# B&R Automation Studio project TD52 (part 56)

#### MsgEMCyclic.st - Cyclic code
```iecst
(*******************************************************************************
Msg_EM	 			 alarms generation MM_emission

This code is confidential and proprietary to the INNIO Company.
It may not be used in any form, or reproduced in any manner,
without written permission of the INNIO Company.
Copyright, INNIO Company, 2023

Customized modifications: -
------------------------

History:
-------
V0.01.0	02.11.2011	lettenb.	new
		27.05.2013	lettenb.	reset OUT_xx.txx2AB.bGnlTripx changed
V4.0.0  02-10-2013  Maxhera,    implementation of the module for modular software
V4.05.0	22.05.2017	Tinello		SCR added, 2276 deleted
		29.01.2018	Tinello		NOx warnings added
V4.05.1	19.02.2018	Tinello		9212 aktiviert, Verzögerung für MS-Sto von 60s auf 10s
V4.07.0	23.04.2019	Tinello		Neue Warnungen für NOx-Selbstdiagnose / Dosierung gestoppt / externe SCR Systeme / NOx lifetime reached
								Warning 2451, 2453 and 3456 can only be acknowledged if blocking of valve/pump is no longer present
								W3482, W3483 und A3380 deleted
V4.07.1	31.10.2019	Tinello		new parameter for lifetime monitoring / measurement signal error delay changed from 10s to 60s
V4.09.0	24.02.2020	Tinello		bugfix -> operating message was too short for HMI / SCR customer input always active
		01.07.2020	Tinello		bugfix -> Message only active if urea dosing controller is active
V4.11.0	11.04.2022	Tinello		CAT temp min monitoring added / W9252 delay from 0->5s
V4.13.0	21.11.2023	Tinello		New operating messages and warnings added
V4.14.0	18.06.2024	Soto	  	Low NOx sensor with CAN communication IF3 considered in W2609 (2023-183)

Instructions for use:
--------------------
1) declare alarm with function block "Alm"
	declare buffert alarm bit bMsg<message number>

2) use template to create a new alarm,
   substitue 0000 by alarm number and make settings:

	xMsg0000.Enable		:=	TRUE;		enable/disable alarm
	xMsg0000.Set		:=	FALSE;		alarm set condition
	xMsg0000.PT			:=	T#0s;		alarm delay time
	xMsg0000.Prio		:=	1;			alarm priority: 1-3 = trip, 4 = warning
	xMsg0000.RiskClass	:=	3;			risk class for remote alarm reset
	xMsg0000.Reset		:=	FALSE;		FALSE: for all standard alarms	prio 1,2,3 and warnings prio 4
										TRUE : for autoreset alarms

	bMsg0000			:=	xMsg0000.Q;	connect buffert alarm bit for VIS and control

3)  expand INIT

3)	include datapoint into OPC configuration for vis

Outstandings:
------------
(*******************************************************************************)
PROGRAM _CYCLIC

	(* reset general trip *)
	OUT_EM.tEM2AB.bGnlTrip1		:=	FALSE;
	OUT_EM.tEM2AB.bGnlTrip2		:=	FALSE;
	OUT_EM.tEM2AB.bGnlTrip3		:=	FALSE;
	OUT_EM.tEM2AB.bGnlWarning	:=	FALSE;
	OUT_EM.tEM2AB.bTriptype1	:=	FALSE;
	OUT_EM.tEM2AB.bTriptype2	:=	FALSE;
	OUT_EM.tEM2AB.bTriptype3	:=	FALSE;

	(* A2276 NOx deviation *) 					(* --> NOT USED *)
	xMsg2276.Enable	   	:= FALSE;
	xMsg2276.Set	   	:= FALSE;
	xMsg2276.PT		   	:= T#0s;
	xMsg2276.Prio 	   	:= 3;
	xMsg2276.RiskClass 	:= 4;
	xMsg2276.Reset		:= FALSE;
	xMsg2276();
	MM2VIS.bMsg2276   	:= xMsg2276.Q;

	(* W2446 SCR BUS communication interrupted *)
	xMsg2446.Enable		:= TRUE;
	xMsg2446.Set		:= bAMM_2446;
	xMsg2446.PT			:= T#10s;
	xMsg2446.Prio		:= 4;
	xMsg2446.RiskClass	:= 4;
	xMsg2446.Reset		:= FALSE;
	xMsg2446();
	MM2VIS.bMsg2446		:= xMsg2446.Q;

	(* W2447 SCR Measuring signal failure urea pressure before dosing *)
	xMsg2447.Enable		:= TRUE;
	xMsg2447.Set		:= bAMM_2447;
	xMsg2447.PT			:= T#10s;
	xMsg2447.Prio		:= 4;
	xMsg2447.RiskClass	:= 4;
	xMsg2447.Reset		:= FALSE;
	xMsg2447();
	MM2VIS.bMsg2447		:= xMsg2447.Q;

	(* W2448 SCR Urea pressure before dosing minimum *)
	xMsg2448.Enable		:= TRUE;
	xMsg2448.Set		:= bAMM_2448;
	xMsg2448.PT			:= T#60s;
	xMsg2448.Prio		:= 4;
	xMsg2448.RiskClass	:= 4;
	xMsg2448.Reset		:= FALSE;
	xMsg2448();
	MM2VIS.bMsg2448		:= xMsg2448.Q;

	(* W2449 SCR Urea pressure before dosing maximum *)
	xMsg2449.Enable		:= TRUE;
	xMsg2449.Set		:= bAMM_2449;
	xMsg2449.PT			:= T#60s;
	xMsg2449.Prio		:= 4;
	xMsg2449.RiskClass	:= 4;
	xMsg2449.Reset		:= FALSE;
	xMsg2449();
	MM2VIS.bMsg2449		:= xMsg2449.Q;

	(* W2450 SCR Leakage in urea dosing cabinet *)
	xMsg2450.Enable		:= Para.bSCR_Active OR Para.bSCR_Cust_Active;
	xMsg2450.Set		:= NOT IN_EM.tLev_SCR_UreaDosingCabinet_Hi.Di;
	xMsg2450.PT			:= T#30s;
	xMsg2450.Prio		:= 4;
	xMsg2450.RiskClass	:= 4;
	xMsg2450.Reset		:= FALSE;
	xMsg2450();
	MM2VIS.bMsg2450		:= xMsg2450.Q;

	(* W2451 SCR Urea dosing valve - error *)
	xMsg2451.Enable		:= TRUE;
	xMsg2451.Set		:= bAMM_2451 OR (MM2VIS.bMsg2451 AND (VIS2MM.bSCR_UreaDosingUnit_Blocked OR
															  VIS2MM.bSCR_UreaDosingUnit2_Blocked  ));
	xMsg2451.PT			:= T#1s;
	xMsg2451.Prio		:= 4;
	xMsg2451.RiskClass	:= 4;
	xMsg2451.Reset		:= FALSE;
	xMsg2451();
	MM2VIS.bMsg2451		:= xMsg2451.Q;

	(* W2452 SCR Measuring signal failure urea flow rate after dosing *)
	xMsg2452.Enable		:= TRUE;
	xMsg2452.Set		:= bAMM_2452;
	xMsg2452.PT			:= T#10s;
	xMsg2452.Prio		:= 4;
	xMsg2452.RiskClass	:= 4;
	xMsg2452.Reset		:= FALSE;
	xMsg2452();
	MM2VIS.bMsg2452		:= xMsg2452.Q;

	(* W2453 SCR Urea flow rate - valve characteristic deviating maximum *)
	xMsg2453.Enable		:= TRUE;
	xMsg2453.Set		:= bAMM_2453 OR (MM2VIS.bMsg2453 AND (VIS2MM.bSCR_UreaDosingUnit_Blocked OR
															  VIS2MM.bSCR_UreaDosingUnit2_Blocked  ));
	xMsg2453.PT			:= T#1s;
	xMsg2453.Prio		:= 4;
	xMsg2453.RiskClass	:= 4;
	xMsg2453.Reset		:= FALSE;
	xMsg2453();
	MM2VIS.bMsg2453		:= xMsg2453.Q;

	(* W2454 SCR Compressed air supply pressure urea injection maximum *)
	xMsg2454.Enable		:= TRUE;
	xMsg2454.Set		:= bAMM_2454;
	xMsg2454.PT			:= T#60s;
	xMsg2454.Prio		:= 4;
	xMsg2454.RiskClass	:= 4;
	xMsg2454.Reset		:= FALSE;
	xMsg2454();
	MM2VIS.bMsg2454		:= xMsg2454.Q;

	(* W2455 SCR Deviation to continous emission monitoring system maximum *)
	xMsg2455.Enable		:= TRUE;
	xMsg2455.Set		:= (EDGEPOS(bAMM_2455_CO) OR EDGEPOS(bAMM_2455_NOx) OR EDGEPOS(bAMM_2455_NOxS)) AND xTON_bRel_SCR_UDC_5m.Q;
	xMsg2455.PT			:= T#0s;
	xMsg2455.Prio		:= 4;
	xMsg2455.RiskClass	:= 4;
	xMsg2455.Reset		:= FALSE;
	xMsg2455();
	MM2VIS.bMsg2455		:= xMsg2455.Q;

	(* W2456 SCR Emission measurement line 1 - O2 maximum *)
	xMsg2456.Enable		:= TRUE;
	xMsg2456.Set		:= bAMM_2456;
	xMsg2456.PT			:= T#60s;
	xMsg2456.Prio		:= 4;
	xMsg2456.RiskClass	:= 4;
	xMsg2456.Reset		:= FALSE;
	xMsg2456();
	MM2VIS.bMsg2456		:= xMsg2456.Q;

	(* W2457 SCR Measuring signal failure emission measurement line 1 - O2 sensor *)
	xMsg2457.Enable		:= TRUE;
	xMsg2457.Set		:= bAMM_2457;
	xMsg2457.PT			:= T#10s;
	xMsg2457.Prio		:= 4;
	xMsg2457.RiskClass	:= 4;
	xMsg2457.Reset		:= FALSE;
	xMsg2457();
	MM2VIS.bMsg2457		:= xMsg2457.Q;

	(* W2458 SCR Measuring signal failure emission measurement line 2 - NO2 sensor *)
	xMsg2458.Enable		:= TRUE;
	xMsg2458.Set		:= bAMM_2458;
	xMsg2458.PT			:= T#10s;
	xMsg2458.Prio		:= 4;
	xMsg2458.RiskClass	:= 4;
	xMsg2458.Reset		:= FALSE;
	xMsg2458();
	MM2VIS.bMsg2458		:= xMsg2458.Q;

	(* W2464 SCR Urea dosing unit (external) - error *)
	xMsg2464.Enable		:= TRUE;
	xMsg2464.Set		:= bAMM_2464;
	xMsg2464.PT			:= T#5s;
	xMsg2464.Prio		:= 4;
	xMsg2464.RiskClass	:= 4;
	xMsg2464.Reset		:= FALSE;
	xMsg2464();
	MM2VIS.bMsg2464		:= xMsg2464.Q;

	(* W2607 CAN failure - NOx sensor CAN interface 1 *)
	xMsg2607.Enable	   	:= TRUE;
	xMsg2607.Set	   	:= bAMM_NOxS_CAN_IF1;
	xMsg2607.PT		   	:= T#10s;
	xMsg2607.Prio 	   	:= 4;
	xMsg2607.RiskClass 	:= 4;
	xMsg2607();
	MM2VIS.bMsg2607    	:= xMsg2607.Q;

	(* W2609 CAN failure - NOx sensor CAN interface 2 or 3 *)
	xMsg2609.Enable	   	:= TRUE;
	xMsg2609.Set	   	:= bAMM_NOxS_CAN_IF2 OR bAMM_NOxS_CAN_IF3;
	xMsg2609.PT		   	:= T#10s;
	xMsg2609.Prio 	   	:= 4;
	xMsg2609.RiskClass 	:= 4;
	xMsg2609();
	MM2VIS.bMsg2609    	:= xMsg2609.Q;

	(* W2610 No connection to the sensor - NOx sensor engine out *)
	xMsg2610.Enable	   	:= TRUE;
	xMsg2610.Set	   	:= bAMM_NOxS_CAN_EngOut;
	xMsg2610.PT		   	:= T#1s;
	xMsg2610.Prio 	   	:= 4;
	xMsg2610.RiskClass 	:= 4;
	xMsg2610();
	MM2VIS.bMsg2610   	:= xMsg2610.Q;

	(* W2697 SCR Urea dosing unit - maintenance needed *)
	xMsg2697.Enable		:= TRUE;
	xMsg2697.Set		:= bAMM_2697;
	xMsg2697.PT			:= T#0s;
	xMsg2697.Prio		:= 4;
	xMsg2697.RiskClass	:= 4;
	xMsg2697.Reset		:= FALSE;
	xMsg2697();
	MM2VIS.bMsg2697		:= xMsg2697.Q;

	(* W2766 Catalyst temperature minimum *)
	xMsg2766.Enable		:= TRUE;
	xMsg2766.Set		:= bAMM_2766;
	xMsg2766.PT			:= T#10s;
	xMsg2766.Prio		:= 4;
	xMsg2766.RiskClass	:= 4;
	xMsg2766.Reset		:= FALSE;
	xMsg2766();
	MM2VIS.bMsg2766		:= xMsg2766.Q;

	(* W2769 SCR Emission measurement air line - moisture maximum *)
	xMsg2769.Enable		:= TRUE;
	xMsg2769.Set		:= bAMM_2769;
	xMsg2769.PT			:= T#0s;
	xMsg2769.Prio		:= 4;
	xMsg2769.RiskClass	:= 4;
	xMsg2769.Reset		:= FALSE;
	xMsg2769();
	MM2VIS.bMsg2769		:= xMsg2769.Q;

	(* A3379 SCR Exhaust temperatures CAT maximum *)
		xTON_T_SCR_Cat3(IN:= NOT IN_EM.tT_SCR_Cat_HiHi.Di, PT:= T#1s);

	xMsg3379.Enable		:= TRUE;
	xMsg3379.Set		:= bAMM_3379 OR xTON_T_SCR_Cat3.Q;
	xMsg3379.PT			:= T#0s;
	xMsg3379.Prio		:= 3;
	xMsg3379.RiskClass	:= 4;
	xMsg3379.Reset		:= FALSE;
	xMsg3379();
	MM2VIS.bMsg3379		:= xMsg3379.Q;

	(* A3380 SCR CO emission average maximum *)			(* --> NOT USED *)
	xMsg3380.Enable		:= FALSE;
	xMsg3380.Set		:= FALSE;
	xMsg3380.PT			:= T#0s;
	xMsg3380.Prio		:= 3;
	xMsg3380.RiskClass	:= 4;
	xMsg3380.Reset		:= FALSE;
	xMsg3380();
	MM2VIS.bMsg3380		:= xMsg3380.Q;

	(* A3381 NOx emissions - short-term average high *)
	xMsg3381.Enable		:= TRUE;
	xMsg3381.Set		:= bAMM_3381;
	xMsg3381.PT			:= T#0s;
	xMsg3381.Prio		:= 3;
	xMsg3381.RiskClass	:= 4;
	xMsg3381.Reset		:= FALSE;
	xMsg3381();
	MM2VIS.bMsg3381		:= xMsg3381.Q;

	(* A3383 SCR Measuring signal failure exhaust temperatures CAT *)
	xMsg3383.Enable		:= TRUE;
	xMsg3383.Set		:= bAMM_3383;
	xMsg3383.PT			:= T#300s;
	xMsg3383.Prio		:= 3;
	xMsg3383.RiskClass	:= 4;
	xMsg3383.Reset		:= FALSE;
	xMsg3383();
	MM2VIS.bMsg3383		:= xMsg3383.Q;

	(*	W3450 SCR Group alarm - exhaust after treatment system *)	(* --> NOT USED *)
	xMsg3450.Enable 	:= FALSE;
	xMsg3450.Set 		:= FALSE;
	xMsg3450.PT			:= T#0s;
	xMsg3450.Prio		:= 4;
	xMsg3450.RiskClass	:= 4;
	xMsg3450();
	MM2VIS.bMsg3450		:= xMsg3450.Q;

	(* W3451 SCR Power supply to the valves interrupted *)
	xMsg3451.Enable		:= TRUE;
	xMsg3451.Set		:= bAMM_3451;
	xMsg3451.PT			:= T#10s;
	xMsg3451.Prio		:= 4;
	xMsg3451.RiskClass	:= 4;
	xMsg3451.Reset		:= FALSE;
	xMsg3451();
	MM2VIS.bMsg3451		:= xMsg3451.Q;

	(* W3452 SCR Measuring signal failure urea pressure after dosing *)
	xMsg3452.Enable		:= TRUE;
	xMsg3452.Set		:= bAMM_3452;
	xMsg3452.PT			:= T#10s;
	xMsg3452.Prio		:= 4;
	xMsg3452.RiskClass	:= 4;
	xMsg3452.Reset		:= FALSE;
	xMsg3452();
	MM2VIS.bMsg3452		:= xMsg3452.Q;

	(* W3453 SCR Urea pressure after dosing maximum *)
	xMsg3453.Enable		:= TRUE;
	xMsg3453.Set		:= bAMM_3453;
	xMsg3453.PT			:= T#0s;
	xMsg3453.Prio		:= 4;
	xMsg3453.RiskClass	:= 4;
	xMsg3453.Reset		:= FALSE;
	xMsg3453();
	MM2VIS.bMsg3453		:= xMsg3453.Q;

	(* W3454 SCR Urea pressure after dosing minimum *)
	xMsg3454.Enable		:= TRUE;
	xMsg3454.Set		:= bAMM_3454;
	xMsg3454.PT			:= T#60s;
	xMsg3454.Prio		:= 4;
	xMsg3454.RiskClass	:= 4;
	xMsg3454.Reset		:= FALSE;
	xMsg3454();
	MM2VIS.bMsg3454		:= xMsg3454.Q;

	(* W3455 SCR Urea flow rate after dosing maximum *)
	xMsg3455.Enable		:= TRUE;
	xMsg3455.Set		:= bAMM_3455;
	xMsg3455.PT			:= T#600s;
	xMsg3455.Prio		:= 4;
	xMsg3455.RiskClass	:= 4;
	xMsg3455.Reset		:= FALSE;
	xMsg3455();
	MM2VIS.bMsg3455		:= xMsg3455.Q;

	(* W3456 SCR Urea dosing pump - error *)
	xMsg3456.Enable		:= TRUE;
	xMsg3456.Set		:= bAMM_3456 OR (MM2VIS.bMsg3456 AND (VIS2MM.bSCR_UreaDosingUnit_Blocked OR
															  VIS2MM.bSCR_UreaDosingUnit2_Blocked  ));
	xMsg3456.PT			:= T#1s;
	xMsg3456.Prio		:= 4;
	xMsg3456.RiskClass	:= 4;
	xMsg3456.Reset		:= FALSE;
	xMsg3456();
	MM2VIS.bMsg3456		:= xMsg3456.Q;

	(* W3457 SCR Urea-air valve blocked *)
	xMsg3457.Enable		:= TRUE;
	xMsg3457.Set		:= bAMM_3457;
	xMsg3457.PT			:= T#45s;
	xMsg3457.Prio		:= 4;
	xMsg3457.RiskClass	:= 4;
	xMsg3457.Reset		:= FALSE;
	xMsg3457();
	MM2VIS.bMsg3457		:= xMsg3457.Q;

	(* W3458 SCR Urea tank level minimum *)
	xMsg3458.Enable		:= Para.bSCR_Active OR Para.bSCR_Cust_Active;
	xMsg3458.Set		:= NOT IN_EM.tLev_SCR_UreaTank_Lo.Di OR (Para.bLev_SCR_UreaTank_Exist AND NOT bAMM_9379 AND IN_EM.tLev_SCR_UreaTank.Ai < Para.rLev_SCR_UreaTank_Lo);
	xMsg3458.PT			:= T#300s;
	xMsg3458.Prio		:= 4;
	xMsg3458.RiskClass	:= 4;
	xMsg3458.Reset		:= FALSE;
	xMsg3458();
	MM2VIS.bMsg3458		:= xMsg3458.Q;

	(* W3459 SCR Urea tank level minimum - dosing deactivated *)
	xMsg3459.Enable		:= TRUE;
	xMsg3459.Set		:= bAMM_3459;
	xMsg3459.PT			:= T#0s;
	xMsg3459.Prio		:= 4;
	xMsg3459.RiskClass	:= 4;
	xMsg3459.Reset		:= FALSE;
	xMsg3459();
	MM2VIS.bMsg3459		:= xMsg3459.Q;

	(* W3460 SCR Urea supply pump not operating *)
	xMsg3460.Enable		:= TRUE;
	xMsg3460.Set		:= bAMM_3460;
	xMsg3460.PT			:= T#30s;
	xMsg3460.Prio		:= 4;
	xMsg3460.RiskClass	:= 4;
	xMsg3460.Reset		:= FALSE;
	xMsg3460();
	MM2VIS.bMsg3460		:= xMsg3460.Q;

	(* W3461 SCR Measuring signal failure compressed air supply pressure urea injection *)
	xMsg3461.Enable		:= TRUE;
	xMsg3461.Set		:= bAMM_3461;
	xMsg3461.PT			:= T#10s;
	xMsg3461.Prio		:= 4;
	xMsg3461.RiskClass	:= 4;
	xMsg3461.Reset		:= FALSE;
	xMsg3461();
	MM2VIS.bMsg3461		:= xMsg3461.Q;

	(* W3462 SCR Compressed air supply pressure urea injection minimum *)
	xMsg3462.Enable		:= TRUE;
	xMsg3462.Set		:= bAMM_3462;
	xMsg3462.PT			:= T#60s;
	xMsg3462.Prio		:= 4;
	xMsg3462.RiskClass	:= 4;
	xMsg3462.Reset		:= FALSE;
	xMsg3462();
	MM2VIS.bMsg3462		:= xMsg3462.Q;

	(* W3463 SCR Compressed air urea injection power supply interrupted *)
	xMsg3463.Enable		:= TRUE;
	xMsg3463.Set		:= bAMM_3463;
	xMsg3463.PT			:= T#10s;
	xMsg3463.Prio		:= 4;
	xMsg3463.RiskClass	:= 4;
	xMsg3463.Reset		:= FALSE;
	xMsg3463();
	MM2VIS.bMsg3463		:= xMsg3463.Q;

	(* W3464 SCR Measuring signal failure exhaust pressure CAT inlet *)
	xMsg3464.Enable		:= TRUE;
	xMsg3464.Set		:= bAMM_3464;
	xMsg3464.PT			:= T#10s;
	xMsg3464.Prio		:= 4;
	xMsg3464.RiskClass	:= 4;
	xMsg3464.Reset		:= FALSE;
	xMsg3464();
	MM2VIS.bMsg3464		:= xMsg3464.Q;

	(* W3465 SCR Measuring signal failure exhaust pressure CAT outlet *)
	xMsg3465.Enable		:= TRUE;
	xMsg3465.Set		:= bAMM_3465;
	xMsg3465.PT			:= T#10s;
	xMsg3465.Prio		:= 4;
	xMsg3465.RiskClass	:= 4;
	xMsg3465.Reset		:= FALSE;
	xMsg3465();
	MM2VIS.bMsg3465		:= xMsg3465.Q;

	(* W3466 SCR Measuring signal failure exhaust temperature CAT inlet *)
	xMsg3466.Enable		:= TRUE;
	xMsg3466.Set		:= bAMM_3466;
	xMsg3466.PT			:= T#10s;
	xMsg3466.Prio		:= 4;
	xMsg3466.RiskClass	:= 4;
	xMsg3466.Reset		:= FALSE;
	xMsg3466();
	MM2VIS.bMsg3466		:= xMsg3466.Q;

	(* W3467 SCR Measuring signal failure exhaust temperature CAT outlet *)
	xMsg3467.Enable		:= TRUE;
	xMsg3467.Set		:= bAMM_3467;
	xMsg3467.PT			:= T#10s;
	xMsg3467.Prio		:= 4;
	xMsg3467.RiskClass	:= 4;
	xMsg3467.Reset		:= FALSE;
	xMsg3467();
	MM2VIS.bMsg3467		:= xMsg3467.Q;

	(* W3469 SCR Exhaust differential pressure CAT maximum *)
	xMsg3469.Enable		:= TRUE;
	xMsg3469.Set		:= bAMM_3469;
	xMsg3469.PT			:= T#300s;
	xMsg3469.Prio		:= 4;
	xMsg3469.RiskClass	:= 4;
	xMsg3469.Reset		:= FALSE;
	xMsg3469();
	MM2VIS.bMsg3469		:= xMsg3469.Q;

	(* W3470 SCR Emission measurement sample gas cooler - error *)
	xMsg3470.Enable		:= TRUE;
	xMsg3470.Set		:= bAMM_3470;
	xMsg3470.PT			:= T#60s;
	xMsg3470.Prio		:= 4;
	xMsg3470.RiskClass	:= 4;
	xMsg3470.Reset		:= FALSE;
	xMsg3470();
	MM2VIS.bMsg3470		:= xMsg3470.Q;

	(* W3471 SCR Emission measurement line 1 - sample gas pump not ready *)
	xMsg3471.Enable		:= TRUE;
	xMsg3471.Set		:= bAMM_3471;
	xMsg3471.PT			:= T#10s;
	xMsg3471.Prio		:= 4;
	xMsg3471.RiskClass	:= 4;
	xMsg3471.Reset		:= FALSE;
	xMsg3471();
	MM2VIS.bMsg3471		:= xMsg3471.Q;

	(* W3472 SCR Emission measurement line 2 - sample gas pump not operating *)
	xMsg3472.Enable		:= TRUE;
	xMsg3472.Set		:= bAMM_3472;
	xMsg3472.PT			:= T#10s;
	xMsg3472.Prio		:= 4;
	xMsg3472.RiskClass	:= 4;
	xMsg3472.Reset		:= FALSE;
	xMsg3472();
	MM2VIS.bMsg3472		:= xMsg3472.Q;

	(* W3473 SCR Emission measurement line 1 - moisture maximum *)
	xMsg3473.Enable		:= TRUE;
	xMsg3473.Set		:= bAMM_3473;
	xMsg3473.PT			:= T#10s;
	xMsg3473.Prio		:= 4;
	xMsg3473.RiskClass	:= 4;
	xMsg3473.Reset		:= FALSE;
	xMsg3473();
	MM2VIS.bMsg3473		:= xMsg3473.Q;

	(* W3474 SCR Emission measurement line 2 - moisture maximum *)
	xMsg3474.Enable		:= TRUE;
	xMsg3474.Set		:= bAMM_3474;
	xMsg3474.PT			:= T#10s;
	xMsg3474.Prio		:= 4;
	xMsg3474.RiskClass	:= 4;
	xMsg3474.Reset		:= FALSE;
	xMsg3474();
	MM2VIS.bMsg3474		:= xMsg3474.Q;

	(* W3475 SCR Emission measurement line 1 - flow rate minimum *)
	xMsg3475.Enable		:= TRUE;
	xMsg3475.Set		:= bAMM_3475;
	xMsg3475.PT			:= T#10s;
	xMsg3475.Prio		:= 4;
	xMsg3475.RiskClass	:= 4;
	xMsg3475.Reset		:= FALSE;
	xMsg3475();
	MM2VIS.bMsg3475		:= xMsg3475.Q;

	(* W3476 SCR Emission measurement line 2 - flow rate minimum *)
	xMsg3476.Enable		:= TRUE;
	xMsg3476.Set		:= bAMM_3476;
	xMsg3476.PT			:= T#10s;
	xMsg3476.Prio		:= 4;
	xMsg3476.RiskClass	:= 4;
	xMsg3476.Reset		:= FALSE;
	xMsg3476();
	MM2VIS.bMsg3476		:= xMsg3476.Q;

	(* W3477 SCR Measuring signal failure emission measurement line 2 - NO sensor *)
	xMsg3477.Enable		:= TRUE;
	xMsg3477.Set		:= bAMM_3477;
	xMsg3477.PT			:= T#10s;
	xMsg3477.Prio		:= 4;
	xMsg3477.RiskClass	:= 4;
	xMsg3477.Reset		:= FALSE;
	xMsg3477();
	MM2VIS.bMsg3477		:= xMsg3477.Q;

	(* W3478 SCR Measuring signal failure emission measurement line 1 - NO sensor *)
	xMsg3478.Enable		:= TRUE;
	xMsg3478.Set		:= bAMM_3478;
	xMsg3478.PT			:= T#10s;
	xMsg3478.Prio		:= 4;
	xMsg3478.RiskClass	:= 4;
	xMsg3478.Reset		:= FALSE;
	xMsg3478();
	MM2VIS.bMsg3478		:= xMsg3478.Q;

	(* W3479 SCR Measuring signal failure emission measurement line 1 - NO2 sensor *)
	xMsg3479.Enable		:= TRUE;
	xMsg3479.Set		:= bAMM_3479;
	xMsg3479.PT			:= T#10s;
	xMsg3479.Prio		:= 4;
	xMsg3479.RiskClass	:= 4;
	xMsg3479.Reset		:= FALSE;
	xMsg3479();
	MM2VIS.bMsg3479		:= xMsg3479.Q;

	(* W3480 SCR NH3 slip detection deactivated *)
	xMsg3480.Enable		:= TRUE;
	xMsg3480.Set		:= bAMM_3480;
	xMsg3480.PT			:= T#0s;
	xMsg3480.Prio		:= 4;
	xMsg3480.RiskClass	:= 4;
	xMsg3480.Reset		:= FALSE;
	xMsg3480();
	MM2VIS.bMsg3480		:= xMsg3480.Q;

	(* W3481 SCR Measuring signal failure emission measurement line 1 - CO sensor *)
	xMsg3481.Enable		:= TRUE;
	xMsg3481.Set		:= bAMM_3481;
	xMsg3481.PT			:= T#10s;
	xMsg3481.Prio		:= 4;
	xMsg3481.RiskClass	:= 4;
	xMsg3481.Reset		:= FALSE;
	xMsg3481();
	MM2VIS.bMsg3481		:= xMsg3481.Q;

	(* W3482 SCR NOx emission to check *)				(* --> NOT USED *)
	xMsg3482.Enable		:= FALSE;
	xMsg3482.Set		:= FALSE;
	xMsg3482.PT			:= T#0s;
	xMsg3482.Prio		:= 4;
	xMsg3482.RiskClass	:= 4;
	xMsg3482.Reset		:= FALSE;
	xMsg3482();
	MM2VIS.bMsg3482		:= xMsg3482.Q;

	(* W3483 SCR CO emission to check *)				(* --> NOT USED *)
	xMsg3483.Enable		:= FALSE;
	xMsg3483.Set		:= FALSE;
	xMsg3483.PT			:= T#0s;
	xMsg3483.Prio		:= 4;
	xMsg3483.RiskClass	:= 4;
	xMsg3483.Reset		:= FALSE;
	xMsg3483();
	MM2VIS.bMsg3483		:= xMsg3483.Q;

	(* W3484 CO emissions - short-term average high *)
	xMsg3484.Enable		:= TRUE;
	xMsg3484.Set		:= bAMM_3484;
	xMsg3484.PT			:= T#0s;
	xMsg3484.Prio		:= 4;
	xMsg3484.RiskClass	:= 4;
	xMsg3484.Reset		:= FALSE;
	xMsg3484();
	MM2VIS.bMsg3484		:= xMsg3484.Q;

	(* W3485 NOx emissions - short-term average high *)
	xMsg3485.Enable		:= TRUE;
	xMsg3485.Set		:= bAMM_3485;
	xMsg3485.PT			:= T#0s;
	xMsg3485.Prio		:= 4;
	xMsg3485.RiskClass	:= 4;
	xMsg3485.Reset		:= FALSE;
	xMsg3485();
	MM2VIS.bMsg3485		:= xMsg3485.Q;

	(* W3486 SCR Urea flow rate after dosing minimum *)
	xMsg3486.Enable		:= TRUE;
	xMsg3486.Set		:= bAMM_3486;
	xMsg3486.PT			:= T#600s;
	xMsg3486.Prio		:= 4;
	xMsg3486.RiskClass	:= 4;
	xMsg3486.Reset		:= FALSE;
	xMsg3486();
	MM2VIS.bMsg3486		:= xMsg3486.Q;

	(* W3487 SCR Exhaust temperature CAT inlet maximum *)
	xMsg3487.Enable		:= TRUE;
	xMsg3487.Set		:= bAMM_3487;
	xMsg3487.PT			:= T#10s;
	xMsg3487.Prio		:= 4;
	xMsg3487.RiskClass	:= 4;
	xMsg3487.Reset		:= FALSE;
	xMsg3487();
	MM2VIS.bMsg3487		:= xMsg3487.Q;

	(* W3488 SCR Exhaust temperature CAT outlet maximum *)
	xMsg3488.Enable		:= TRUE;
	xMsg3488.Set		:= bAMM_3488;
	xMsg3488.PT			:= T#10s;
	xMsg3488.Prio		:= 4;
	xMsg3488.RiskClass	:= 4;
	xMsg3488.Reset		:= FALSE;
	xMsg3488();
	MM2VIS.bMsg3488		:= xMsg3488.Q;

	(* W3489 SCR Emergency Stop SCR control cabinet *)		(* --> NOT USED	*)
	xMsg3489.Enable 	:= FALSE;
	xMsg3489.Set 		:= FALSE;
	xMsg3489.PT			:= T#0s;
	xMsg3489.Prio		:= 4;
	xMsg3489.RiskClass	:= 4;
	xMsg3489.Reset		:= FALSE;
	xMsg3489();
	MM2VIS.bMsg3489		:= xMsg3489.Q;

	(* W9201 Measuring signal failure O2, NOx sensor engine out *)
	xMsg9201.Enable 	:= TRUE;
	xMsg9201.Set 		:= bAMM_O2_NOxS_EngOut_Ms;
	xMsg9201.PT			:= T#60s;
	xMsg9201.Prio		:= 4;
	xMsg9201.RiskClass	:= 4;
	xMsg9201.Reset		:= FALSE;
	xMsg9201();
	MM2VIS.bMsg9201		:= xMsg9201.Q;

	(* W9202 Measuring signal failure NOx, NOx sensor engine out *)
	xMsg9202.Enable 	:= TRUE;
	xMsg9202.Set 		:= bAMM_NOx_NOxS_EngOut_Ms;
	xMsg9202.PT			:= T#60s;
	xMsg9202.Prio		:= 4;
	xMsg9202.RiskClass	:= 4;
	xMsg9202.Reset		:= FALSE;
	xMsg9202();
	MM2VIS.bMsg9202		:= xMsg9202.Q;

	(* W9203 No connection to the sensor - NOx sensor engine out A *)
	xMsg9203.Enable 	:= TRUE;
	xMsg9203.Set 		:= bAMM_NOxS_CAN_EngOut_A;
	xMsg9203.PT			:= T#1s;
	xMsg9203.Prio		:= 4;
	xMsg9203.RiskClass	:= 4;
	xMsg9203.Reset		:= FALSE;
	xMsg9203();
	MM2VIS.bMsg9203		:= xMsg9203.Q;

	(* W9204 Measuring signal failure O2, NOx sensor engine out – bank A *)
	xMsg9204.Enable 	:= TRUE;
	xMsg9204.Set 		:= bAMM_O2_NOxS_EngOut_A_Ms;
	xMsg9204.PT			:= T#60s;
	xMsg9204.Prio		:= 4;
	xMsg9204.RiskClass	:= 4;
	xMsg9204.Reset		:= FALSE;
	xMsg9204();
	MM2VIS.bMsg9204		:= xMsg9204.Q;

	(* W9205 Measuring signal failure NOx, NOx sensor engine out – bank A *)
	xMsg9205.Enable 	:= TRUE;
	xMsg9205.Set 		:= bAMM_NOx_NOxS_EngOut_A_Ms;
	xMsg9205.PT			:= T#60s;
	xMsg9205.Prio		:= 4;
	xMsg9205.RiskClass	:= 4;
	xMsg9205.Reset		:= FALSE;
	xMsg9205();
	MM2VIS.bMsg9205		:= xMsg9205.Q;

	(* W9206 No connection to the sensor - NOx sensor engine out B *)
	xMsg9206.Enable 	:= TRUE;
	xMsg9206.Set 		:= bAMM_NOxS_CAN_EngOut_B;
	xMsg9206.PT			:= T#1s;
	xMsg9206.Prio		:= 4;
	xMsg9206.RiskClass	:= 4;
	xMsg9206.Reset		:= FALSE;
	xMsg9206();
	MM2VIS.bMsg9206		:= xMsg9206.Q;

	(* W9207 Measuring signal failure O2, NOx sensor engine out – bank B *)
	xMsg9207.Enable 	:= TRUE;
	xMsg9207.Set 		:= bAMM_O2_NOxS_EngOut_B_Ms;
	xMsg9207.PT			:= T#60s;
	xMsg9207.Prio		:= 4;
	xMsg9207.RiskClass	:= 4;
	xMsg9207.Reset		:= FALSE;
	xMsg9207();
	MM2VIS.bMsg9207		:= xMsg9207.Q;

	(* W9208 Measuring signal failure NOx, NOx sensor engine out – bank B *)
	xMsg9208.Enable 	:= TRUE;
	xMsg9208.Set 		:= bAMM_NOx_NOxS_EngOut_B_Ms;
	xMsg9208.PT			:= T#60s;
	xMsg9208.Prio		:= 4;
	xMsg9208.RiskClass	:= 4;
	xMsg9208.Reset		:= FALSE;
	xMsg9208();
	MM2VIS.bMsg9208		:= xMsg9208.Q;

	(* W9209 No connection to the sensor - NOx sensor CAT out *)
	xMsg9209.Enable 	:= TRUE;
	xMsg9209.Set 		:= bAMM_NOxS_CAN_CatOut;
	xMsg9209.PT			:= T#1s;
	xMsg9209.Prio		:= 4;
	xMsg9209.RiskClass	:= 4;
	xMsg9209.Reset		:= FALSE;
	xMsg9209();
	MM2VIS.bMsg9209		:= xMsg9209.Q;

	(* W9210 Measuring signal failure O2, NOx sensor CAT out *)
	xMsg9210.Enable 	:= TRUE;
	xMsg9210.Set 		:= bAMM_O2_NOxS_CatOut_Ms;
	xMsg9210.PT			:= T#60s;
	xMsg9210.Prio		:= 4;
	xMsg9210.RiskClass	:= 4;
	xMsg9210.Reset		:= FALSE;
	xMsg9210();
	MM2VIS.bMsg9210		:= xMsg9210.Q;

	(* W9211 Measuring signal failure NOx, NOx sensor CAT out *)
	xMsg9211.Enable 	:= TRUE;
	xMsg9211.Set 		:= bAMM_NOx_NOxS_CatOut_Ms;
	xMsg9211.PT			:= T#60s;
	xMsg9211.Prio		:= 4;
	xMsg9211.RiskClass	:= 4;
	xMsg9211.Reset		:= FALSE;
	xMsg9211();
	MM2VIS.bMsg9211		:= xMsg9211.Q;

	(* W9212 SCR Air compressor - maintenance needed  *)
	xMsg9212.Enable 	:= TRUE;
	xMsg9212.Set 		:= bAMM_9212;
	xMsg9212.PT			:= T#0s;
	xMsg9212.Prio		:= 4;
	xMsg9212.RiskClass	:= 4;
	xMsg9212.Reset		:= FALSE;
	xMsg9212();
	MM2VIS.bMsg9212		:= xMsg9212.Q;

	(* W9233 Lifetime reached - NOx sensor engine out *)
	xMsg9233.Enable 	:= TRUE;
	xMsg9233.Set 		:= bNOxS_EngOut_Exist 	AND MM2VIS.iNOxS_EngOut_OpHours   >= Para.iNOxS_Lifetime;
	xMsg9233.PT			:= T#0s;
	xMsg9233.Prio		:= 4;
	xMsg9233.RiskClass	:= 4;
	xMsg9233.Reset		:= FALSE;
	xMsg9233();
	MM2VIS.bMsg9233		:= xMsg9233.Q;

	(* W9234 Lifetime reached - NOx sensor engine out A *)
	xMsg9234.Enable 	:= TRUE;
	xMsg9234.Set 		:= bNOxS_EngOut_A_Exist AND MM2VIS.iNOxS_EngOut_A_OpHours >= Para.iNOxS_Lifetime;
	xMsg9234.PT			:= T#0s;
	xMsg9234.Prio		:= 4;
	xMsg9234.RiskClass	:= 4;
	xMsg9234.Reset		:= FALSE;
	xMsg9234();
	MM2VIS.bMsg9234		:= xMsg9234.Q;

	(* W9235 Lifetime reached - NOx sensor engine out B *)
	xMsg9235.Enable 	:= TRUE;
	xMsg9235.Set 		:= bNOxS_EngOut_B_Exist	AND MM2VIS.iNOxS_EngOut_B_OpHours >= Para.iNOxS_Lifetime;
	xMsg9235.PT			:= T#0s;
	xMsg9235.Prio		:= 4;
	xMsg9235.RiskClass	:= 4;
	xMsg9235.Reset		:= FALSE;
	xMsg9235();
	MM2VIS.bMsg9235		:= xMsg9235.Q;

	(* W9236 Lifetime reached - NOx sensor CAT out *)
	xMsg9236.Enable 	:= TRUE;
	xMsg9236.Set 		:= bNOxS_CatOut_Exist 	AND MM2VIS.iNOxS_CatOut_OpHours   >= Para.iNOxS_Lifetime;
	xMsg9236.PT			:= T#0s;
	xMsg9236.Prio		:= 4;
	xMsg9236.RiskClass	:= 4;
	xMsg9236.Reset		:= FALSE;
	xMsg9236();
	MM2VIS.bMsg9236		:= xMsg9236.Q;

	(* W9250 O2 deviation bank A/B maximum - NOx sensor engine out *)
	xMsg9250.Enable 	:= TRUE;
	xMsg9250.Set 		:= bAMM_O2_NOxS_EngOut_Dev_Hi;
	xMsg9250.PT			:= T#0s;
	xMsg9250.Prio		:= 4;
	xMsg9250.RiskClass	:= 4;
	xMsg9250.Reset		:= FALSE;
	xMsg9250();
	MM2VIS.bMsg9250		:= xMsg9250.Q;

	(* W9251 NOx deviation bank A/B maximum - NOx sensor engine out *)
	xMsg9251.Enable 	:= TRUE;
	xMsg9251.Set 		:= bAMM_NOx_NOxS_EngOut_Dev_Hi;
	xMsg9251.PT			:= T#0s;
	xMsg9251.Prio		:= 4;
	xMsg9251.RiskClass	:= 4;
	xMsg9251.Reset		:= FALSE;
	xMsg9251();
	MM2VIS.bMsg9251		:= xMsg9251.Q;

	(* W9252 NOx emissions - daily average high *)
	xMsg9252.Enable 	:= TRUE;
	xMsg9252.Set 		:= bAMM_NOx_Em_AvgDaily_Hi;
	xMsg9252.PT			:= T#5s;
	xMsg9252.Prio		:= 4;
	xMsg9252.RiskClass	:= 4;
	xMsg9252.Reset		:= FALSE;
	xMsg9252();
	MM2VIS.bMsg9252		:= xMsg9252.Q;

	(* W9277 SCR Urea dosing stopped - error *)
	xMsg9277.Enable 	:= TRUE;
	xMsg9277.Set 		:= bAMM_9277;
	xMsg9277.PT			:= T#0s;
	xMsg9277.Prio		:= 4;
	xMsg9277.RiskClass	:= 4;
	xMsg9277.Reset		:= FALSE;
	xMsg9277();
	MM2VIS.bMsg9277		:= xMsg9277.Q;

	(* W9278 SCR Catalyst - failure (DI from customer) *)
	xMsg9278.Enable 	:= TRUE;
	xMsg9278.Set 		:= NOT IN_EM.tSCR_Catalyst_Rdy.Di;
	xMsg9278.PT			:= T#1s;
	xMsg9278.Prio		:= 4;
	xMsg9278.RiskClass	:= 4;
	xMsg9278.Reset		:= FALSE;
	xMsg9278();
	MM2VIS.bMsg9278		:= xMsg9278.Q;

	(* W9379 SCR Measuring signal failure urea tank level *)
	xMsg9379.Enable 	:= TRUE;
	xMsg9379.Set 		:= bAMM_9379;
	xMsg9379.PT			:= T#10s;
	xMsg9379.Prio		:= 4;
	xMsg9379.RiskClass	:= 4;
	xMsg9379.Reset		:= FALSE;
	xMsg9379();
	MM2VIS.bMsg9379		:= xMsg9379.Q;

	(* W9380 SCR Urea flow dosing error *)
	xMsg9380.Enable 	:= TRUE;
	xMsg9380.Set 		:= bAMM_9380;
	xMsg9380.PT			:= T#0s;
	xMsg9380.Prio		:= 4;
	xMsg9380.RiskClass	:= 4;
	xMsg9380.Reset		:= FALSE;
	xMsg9380();
	MM2VIS.bMsg9380		:= xMsg9380.Q;

	(*---------------------------------------------------------------------------*)
	(* operating messages > AMM *)

	(* B2877 SCR Exhaust after treatment deactivated *)	(* --> NOT USED *)
	xMsg2877.Enable 	:= FALSE;
	xMsg2877.Set 		:= FALSE;
	xMsg2877.Reset     	:= TRUE;
	xMsg2877();
	MM2VIS.bMsg2877		:= xMsg2877.Q;

	(* B2878 SCR Urea dosing activated *)
	xMsg2878.Enable		:= TRUE;
	xMsg2878.Set		:= bOpM_2878;
	xMsg2878.Reset		:= TRUE;
	xMsg2878();
	MM2VIS.bMsg2878		:= xMsg2878.Q;

	(* B2879 SCR Urea dosing deactivated *)
	xMsg2879.Enable		:= TRUE;
	xMsg2879.Set		:= bOpM_2879;
	xMsg2879.Reset		:= TRUE;
	xMsg2879();
	MM2VIS.bMsg2879		:= xMsg2879.Q;

	(* B2884 SCR Manual mode on *)
	xMsg2884.Enable		:= TRUE;
	xMsg2884.Set		:= bOpM_2884;
	xMsg2884.Reset		:= TRUE;
	xMsg2884();
	MM2VIS.bMsg2884		:= xMsg2884.Q;

	(* B2885 SCR Manual mode off *)
	xMsg2885.Enable		:= TRUE;
	xMsg2885.Set		:= bOpM_2885;
	xMsg2885.Reset		:= TRUE;
	xMsg2885();
	MM2VIS.bMsg2885		:= xMsg2885.Q;

	(* B2923 SCR NH3 slip detection started *)
	xMsg2923.Enable		:= TRUE;
	xMsg2923.Set		:= bOpM_2923;
	xMsg2923.Reset		:= TRUE;
	xMsg2923();
	MM2VIS.bMsg2923		:= xMsg2923.Q;

	(* B2924 SCR NH3 slip detection completed *)
	xMsg2924.Enable		:= TRUE;
	xMsg2924.Set		:= bOpM_2924;
	xMsg2924.Reset		:= TRUE;
	xMsg2924();
	MM2VIS.bMsg2924		:= xMsg2924.Q;

	(* B2971 Error during self-diagnosis - NOx sensor engine out *)
	xTOF_EngOut_DiagErr(IN 	:= bOpM_NOxS_EngOut_DiagErr, 	PT := T#1s);		(* increase message time from 100ms to 1s for HMI *)

	xMsg2971.Enable			:= TRUE;
	xMsg2971.Set			:= xTOF_EngOut_DiagErr.Q;
	xMsg2971.Reset			:= TRUE;
	xMsg2971();
	MM2VIS.bMsg2971			:= xMsg2971.Q;

	(* B2974 Error during self-diagnosis - NOx sensor engine out A *)
	xTOF_EngOut_A_DiagErr(IN:= bOpM_NOxS_EngOut_A_DiagErr, 	PT := T#1s);		(* increase message time from 100ms to 1s for HMI *)

	xMsg2974.Enable			:= TRUE;
	xMsg2974.Set			:= xTOF_EngOut_A_DiagErr.Q;
	xMsg2974.Reset			:= TRUE;
	xMsg2974();
	MM2VIS.bMsg2974			:= xMsg2974.Q;

	(* B2977 Error during self-diagnosis - NOx sensor engine out B *)
	xTOF_EngOut_B_DiagErr(IN:= bOpM_NOxS_EngOut_B_DiagErr, 	PT := T#1s);		(* increase message time from 100ms to 1s for HMI *)

	xMsg2977.Enable			:= TRUE;
	xMsg2977.Set			:= xTOF_EngOut_B_DiagErr.Q;
	xMsg2977.Reset			:= TRUE;
	xMsg2977();
	MM2VIS.bMsg2977			:= xMsg2977.Q;

	(* B2980 Error during self-diagnosis - NOx sensor CAT out *)
	xTOF_CatOut_DiagErr(IN 	:= bOpM_NOxS_CatOut_DiagErr, 	PT := T#1s);		(* increase message time from 100ms to 1s for HMI *)

	xMsg2980.Enable			:= TRUE;
	xMsg2980.Set			:= xTOF_CatOut_DiagErr.Q;
	xMsg2980.Reset			:= TRUE;
	xMsg2980();
	MM2VIS.bMsg2980			:= xMsg2980.Q;

	(* B9077 SCR NH3 slip detection interrupted *)
	xMsg9077.Enable			:= TRUE;
	xMsg9077.Set			:= bOpM_9077;
	xMsg9077.Reset			:= TRUE;
	xMsg9077();
	MM2VIS.bMsg9077			:= xMsg9077.Q;

	(* B9079 SCR Urea dosing - dosing conditions reached *)
	xMsg9079.Enable			:= TRUE;
	xMsg9079.Set			:= bOpM_9079;
	xMsg9079.Reset			:= TRUE;
	xMsg9079();
	MM2VIS.bMsg9079			:= xMsg9079.Q;

	(* B9080 SCR Urea dosing - dosing conditions ended *)
	xMsg9080.Enable			:= TRUE;
	xMsg9080.Set			:= bOpM_9080;
	xMsg9080.Reset			:= TRUE;
	xMsg9080();
	MM2VIS.bMsg9080			:= xMsg9080.Q;

	(* B9081 SCR Urea dosing - requested *)
	xMsg9081.Enable			:= TRUE;
	xMsg9081.Set			:= bOpM_9081;
	xMsg9081.Reset			:= TRUE;
	xMsg9081();
	MM2VIS.bMsg9081			:= xMsg9081.Q;

	(* B9082 SCR Urea dosing - unrequested *)
	xMsg9082.Enable			:= TRUE;
	xMsg9082.Set			:= bOpM_9082;
	xMsg9082.Reset			:= TRUE;
	xMsg9082();
	MM2VIS.bMsg9082			:= xMsg9082.Q;

	(*--------------------------------------------------------------------------*)
	(* general alarms for further module operations *)
	bGnlTrip1	:= OUT_EM.tEM2AB.bGnlTrip1   OR IN_EM.tAB2EM.bGnlTrip1;
	bGnlTrip2	:= OUT_EM.tEM2AB.bGnlTrip2   OR IN_EM.tAB2EM.bGnlTrip2;
	bGnlTrip3	:= OUT_EM.tEM2AB.bGnlTrip3   OR IN_EM.tAB2EM.bGnlTrip3;
	bGnlWarning	:= OUT_EM.tEM2AB.bGnlWarning OR IN_EM.tAB2EM.bGnlWarning;

	bGnlTrip	:=	bGnlTrip1 OR bGnlTrip2 OR bGnlTrip3;

	(*******************************************************************************)
END_PROGRAM
```

#### MsgEMInit.st - Initial code
```iecst
(*******************************************************************************
Msg_EM	 			 alarms generation MM_emission

This code is confidential and proprietary to the INNIO Company.
It may not be used in any form, or reproduced in any manner,
without written permission of the INNIO Company.
Copyright, INNIO Company, 2019

Customized modifications: -
------------------------

History:
-------
V0.00.0	29.07.2011	lettenb.	new
V4.00.0 22-08-2013  Maxhera,    implementation of the module for modular software
V4.05.0	22.05.2017	Tinello		SCR added
		29.01.2018	Tinello		NOx warnings added

Instructions for use:
--------------------
1) declare alarm with function block "Msg"

2) use template to create a new alarm, substitue 0000 by message number:

	xMsg0000.Num		:=	0000;					alarm number
	xMsg0000.AmmSysAdr	:=  iAdrAmmBase2MM;			do not change
	xMsg0000.AmmOutAdr	:=  iAdrMM2AmmBase;			do not change

3) 	set alarm number

Outstandings:
------------
(*******************************************************************************)
PROGRAM _INIT

	iAdrAmmBase2MM		:=  ADR(IN_EM.tAB2EM);
	iAdrMM2AmmBase		:=  ADR(OUT_EM.tEM2AB);

	xMsg2276.Num		:= 2276;
	xMsg2276.AmmInAdr	:=  iAdrAmmBase2MM;
	xMsg2276.AmmOutAdr	:=  iAdrMM2AmmBase;

	xMsg2446.Num		:= 2446;
	xMsg2446.AmmInAdr	:= iAdrAmmBase2MM;
	xMsg2446.AmmOutAdr	:= iAdrMM2AmmBase;

	xMsg2447.Num		:= 2447;
	xMsg2447.AmmInAdr	:= iAdrAmmBase2MM;
	xMsg2447.AmmOutAdr	:= iAdrMM2AmmBase;

	xMsg2448.Num		:= 2448;
	xMsg2448.AmmInAdr	:= iAdrAmmBase2MM;
	xMsg2448.AmmOutAdr	:= iAdrMM2AmmBase;

	xMsg2449.Num		:= 2449;
	xMsg2449.AmmInAdr	:= iAdrAmmBase2MM;
	xMsg2449.AmmOutAdr	:= iAdrMM2AmmBase;

	xMsg2450.Num		:= 2450;
	xMsg2450.AmmInAdr	:= iAdrAmmBase2MM;
	xMsg2450.AmmOutAdr	:= iAdrMM2AmmBase;

	xMsg2451.Num		:= 2451;
	xMsg2451.AmmInAdr	:= iAdrAmmBase2MM;
	xMsg2451.AmmOutAdr	:= iAdrMM2AmmBase;

	xMsg2452.Num		:= 2452;
	xMsg2452.AmmInAdr	:= iAdrAmmBase2MM;
	xMsg2452.AmmOutAdr	:= iAdrMM2AmmBase;

	xMsg2453.Num		:= 2453;
	xMsg2453.AmmInAdr	:= iAdrAmmBase2MM;
	xMsg2453.AmmOutAdr	:= iAdrMM2AmmBase;

	xMsg2454.Num		:= 2454;
	xMsg2454.AmmInAdr	:= iAdrAmmBase2MM;
	xMsg2454.AmmOutAdr	:= iAdrMM2AmmBase;

	xMsg2455.Num		:= 2455;
	xMsg2455.AmmInAdr	:= iAdrAmmBase2MM;
	xMsg2455.AmmOutAdr	:= iAdrMM2AmmBase;

	xMsg2456.Num		:= 2456;
	xMsg2456.AmmInAdr	:= iAdrAmmBase2MM;
	xMsg2456.AmmOutAdr	:= iAdrMM2AmmBase;

	xMsg2457.Num		:= 2457;
	xMsg2457.AmmInAdr	:= iAdrAmmBase2MM;
	xMsg2457.AmmOutAdr	:= iAdrMM2AmmBase;

	xMsg2458.Num		:= 2458;
	xMsg2458.AmmInAdr	:= iAdrAmmBase2MM;
	xMsg2458.AmmOutAdr	:= iAdrMM2AmmBase;

	xMsg2464.Num		:= 2464;
	xMsg2464.AmmInAdr	:= iAdrAmmBase2MM;
	xMsg2464.AmmOutAdr	:= iAdrMM2AmmBase;

	xMsg2607.Num		:= 2607;
	xMsg2607.AmmInAdr	:= iAdrAmmBase2MM;
	xMsg2607.AmmOutAdr	:= iAdrMM2AmmBase;

	xMsg2609.Num		:= 2609;
	xMsg2609.AmmInAdr	:= iAdrAmmBase2MM;
	xMsg2609.AmmOutAdr	:=  iAdrMM2AmmBase;

	xMsg2610.Num		:= 2610;
	xMsg2610.AmmInAdr	:=  iAdrAmmBase2MM;
	xMsg2610.AmmOutAdr	:=  iAdrMM2AmmBase;

	xMsg2697.Num		:=	2697;
	xMsg2697.AmmInAdr	:=  iAdrAmmBase2MM;
	xMsg2697.AmmOutAdr	:=  iAdrMM2AmmBase;

	xMsg2766.Num		:=	2766;
	xMsg2766.AmmInAdr	:=  iAdrAmmBase2MM;
	xMsg2766.AmmOutAdr	:=  iAdrMM2AmmBase;

	xMsg2769.Num		:=	2769;
	xMsg2769.AmmInAdr	:=  iAdrAmmBase2MM;
	xMsg2769.AmmOutAdr	:=  iAdrMM2AmmBase;

	xMsg2877.Num 		:= 2877;
	xMsg2877.AmmInAdr	:= iAdrAmmBase2MM;
	xMsg2877.AmmOutAdr	:= iAdrMM2AmmBase;

	xMsg2878.Num 		:= 2878;
	xMsg2878.AmmInAdr	:= iAdrAmmBase2MM;
	xMsg2878.AmmOutAdr	:= iAdrMM2AmmBase;

	xMsg2879.Num 		:= 2879;
	xMsg2879.AmmInAdr	:= iAdrAmmBase2MM;
	xMsg2879.AmmOutAdr	:= iAdrMM2AmmBase;

	xMsg2884.Num 		:= 2884;
	xMsg2884.AmmInAdr	:= iAdrAmmBase2MM;
	xMsg2884.AmmOutAdr	:= iAdrMM2AmmBase;

	xMsg2885.Num 		:= 2885;
	xMsg2885.AmmInAdr	:= iAdrAmmBase2MM;
	xMsg2885.AmmOutAdr	:= iAdrMM2AmmBase;

	xMsg2923.Num 		:= 2923;
	xMsg2923.AmmInAdr	:= iAdrAmmBase2MM;
	xMsg2923.AmmOutAdr	:= iAdrMM2AmmBase;

	xMsg2924.Num 		:= 2924;
	xMsg2924.AmmInAdr	:= iAdrAmmBase2MM;
	xMsg2924.AmmOutAdr	:= iAdrMM2AmmBase;

	xMsg2971.Num 		:= 2971;
	xMsg2971.AmmInAdr	:= iAdrAmmBase2MM;
	xMsg2971.AmmOutAdr	:= iAdrMM2AmmBase;

	xMsg2974.Num 		:= 2974;
	xMsg2974.AmmInAdr	:= iAdrAmmBase2MM;
	xMsg2974.AmmOutAdr	:= iAdrMM2AmmBase;

	xMsg2977.Num 		:= 2977;
	xMsg2977.AmmInAdr	:= iAdrAmmBase2MM;
	xMsg2977.AmmOutAdr	:= iAdrMM2AmmBase;

	xMsg2980.Num 		:= 2980;
	xMsg2980.AmmInAdr	:= iAdrAmmBase2MM;
	xMsg2980.AmmOutAdr	:= iAdrMM2AmmBase;

	xMsg3379.Num 		:= 3379;
	xMsg3379.AmmInAdr	:= iAdrAmmBase2MM;
	xMsg3379.AmmOutAdr	:= iAdrMM2AmmBase;

	xMsg3380.Num 		:= 3380;
	xMsg3380.AmmInAdr	:= iAdrAmmBase2MM;
	xMsg3380.AmmOutAdr	:= iAdrMM2AmmBase;

	xMsg3381.Num 		:= 3381;
	xMsg3381.AmmInAdr	:= iAdrAmmBase2MM;
	xMsg3381.AmmOutAdr	:= iAdrMM2AmmBase;

	xMsg3383.Num 		:= 3383;
	xMsg3383.AmmInAdr	:= iAdrAmmBase2MM;
	xMsg3383.AmmOutAdr	:= iAdrMM2AmmBase;

	xMsg3450.Num 		:= 3450;
	xMsg3450.AmmInAdr	:= iAdrAmmBase2MM;
	xMsg3450.AmmOutAdr	:= iAdrMM2AmmBase;

	xMsg3451.Num 		:= 3451;
	xMsg3451.AmmInAdr	:= iAdrAmmBase2MM;
	xMsg3451.AmmOutAdr	:= iAdrMM2AmmBase;

	xMsg3452.Num 		:= 3452;
	xMsg3452.AmmInAdr	:= iAdrAmmBase2MM;
	xMsg3452.AmmOutAdr	:= iAdrMM2AmmBase;

	xMsg3453.Num 		:= 3453;
	xMsg3453.AmmInAdr	:= iAdrAmmBase2MM;
	xMsg3453.AmmOutAdr	:= iAdrMM2AmmBase;

	xMsg3454.Num 		:= 3454;
	xMsg3454.AmmInAdr	:= iAdrAmmBase2MM;
	xMsg3454.AmmOutAdr	:= iAdrMM2AmmBase;

	xMsg3455.Num 		:= 3455;
	xMsg3455.AmmInAdr	:= iAdrAmmBase2MM;
	xMsg3455.AmmOutAdr	:= iAdrMM2AmmBase;

	xMsg3456.Num 		:= 3456;
	xMsg3456.AmmInAdr	:= iAdrAmmBase2MM;
	xMsg3456.AmmOutAdr	:= iAdrMM2AmmBase;

	xMsg3457.Num 		:= 3457;
	xMsg3457.AmmInAdr	:= iAdrAmmBase2MM;
	xMsg3457.AmmOutAdr	:= iAdrMM2AmmBase;

	xMsg3458.Num 		:= 3458;
	xMsg3458.AmmInAdr	:= iAdrAmmBase2MM;
	xMsg3458.AmmOutAdr	:= iAdrMM2AmmBase;

	xMsg3459.Num 		:= 3459;
	xMsg3459.AmmInAdr	:= iAdrAmmBase2MM;
	xMsg3459.AmmOutAdr	:= iAdrMM2AmmBase;

	xMsg3460.Num 		:= 3460;
	xMsg3460.AmmInAdr	:= iAdrAmmBase2MM;
	xMsg3460.AmmOutAdr	:= iAdrMM2AmmBase;

	xMsg3461.Num 		:= 3461;
	xMsg3461.AmmInAdr	:= iAdrAmmBase2MM;
	xMsg3461.AmmOutAdr	:= iAdrMM2AmmBase;

	xMsg3462.Num 		:= 3462;
	xMsg3462.AmmInAdr	:= iAdrAmmBase2MM;
	xMsg3462.AmmOutAdr	:= iAdrMM2AmmBase;

	xMsg3463.Num 		:= 3463;
	xMsg3463.AmmInAdr	:= iAdrAmmBase2MM;
	xMsg3463.AmmOutAdr	:= iAdrMM2AmmBase;

	xMsg3464.Num 		:= 3464;
	xMsg3464.AmmInAdr	:= iAdrAmmBase2MM;
	xMsg3464.AmmOutAdr	:= iAdrMM2AmmBase;

	xMsg3465.Num 		:= 3465;
	xMsg3465.AmmInAdr	:= iAdrAmmBase2MM;
	xMsg3465.AmmOutAdr	:= iAdrMM2AmmBase;

	xMsg3466.Num 		:= 3466;
	xMsg3466.AmmInAdr	:= iAdrAmmBase2MM;
	xMsg3466.AmmOutAdr	:= iAdrMM2AmmBase;

	xMsg3467.Num 		:= 3467;
	xMsg3467.AmmInAdr	:= iAdrAmmBase2MM;
	xMsg3467.AmmOutAdr	:= iAdrMM2AmmBase;

	xMsg3469.Num 		:= 3469;
	xMsg3469.AmmInAdr	:= iAdrAmmBase2MM;
	xMsg3469.AmmOutAdr	:= iAdrMM2AmmBase;

	xMsg3470.Num 		:= 3470;
	xMsg3470.AmmInAdr	:= iAdrAmmBase2MM;
	xMsg3470.AmmOutAdr	:= iAdrMM2AmmBase;

	xMsg3471.Num 		:= 3471;
	xMsg3471.AmmInAdr	:= iAdrAmmBase2MM;
	xMsg3471.AmmOutAdr	:= iAdrMM2AmmBase;

	xMsg3472.Num 		:= 3472;
	xMsg3472.AmmInAdr	:= iAdrAmmBase2MM;
	xMsg3472.AmmOutAdr	:= iAdrMM2AmmBase;

	xMsg3473.Num 		:= 3473;
	xMsg3473.AmmInAdr	:= iAdrAmmBase2MM;
	xMsg3473.AmmOutAdr	:= iAdrMM2AmmBase;

	xMsg3474.Num 		:= 3474;
	xMsg3474.AmmInAdr	:= iAdrAmmBase2MM;
	xMsg3474.AmmOutAdr	:= iAdrMM2AmmBase;

	xMsg3475.Num 		:= 3475;
	xMsg3475.AmmInAdr	:= iAdrAmmBase2MM;
	xMsg3475.AmmOutAdr	:= iAdrMM2AmmBase;

	xMsg3476.Num 		:= 3476;
	xMsg3476.AmmInAdr	:= iAdrAmmBase2MM;
	xMsg3476.AmmOutAdr	:= iAdrMM2AmmBase;

	xMsg3477.Num 		:= 3477;
	xMsg3477.AmmInAdr	:= iAdrAmmBase2MM;
	xMsg3477.AmmOutAdr	:= iAdrMM2AmmBase;

	xMsg3478.Num 		:= 3478;
	xMsg3478.AmmInAdr	:= iAdrAmmBase2MM;
	xMsg3478.AmmOutAdr	:= iAdrMM2AmmBase;

	xMsg3479.Num 		:= 3479;
	xMsg3479.AmmInAdr	:= iAdrAmmBase2MM;
	xMsg3479.AmmOutAdr	:= iAdrMM2AmmBase;

	xMsg3480.Num 		:= 3480;
	xMsg3480.AmmInAdr	:= iAdrAmmBase2MM;
	xMsg3480.AmmOutAdr	:= iAdrMM2AmmBase;

	xMsg3481.Num 		:= 3481;
	xMsg3481.AmmInAdr	:= iAdrAmmBase2MM;
	xMsg3481.AmmOutAdr	:= iAdrMM2AmmBase;

	xMsg3482.Num 		:= 3482;
	xMsg3482.AmmInAdr	:= iAdrAmmBase2MM;
	xMsg3482.AmmOutAdr	:= iAdrMM2AmmBase;

	xMsg3483.Num 		:= 3483;
	xMsg3483.AmmInAdr	:= iAdrAmmBase2MM;
	xMsg3483.AmmOutAdr	:= iAdrMM2AmmBase;

	xMsg3484.Num 		:= 3484;
	xMsg3484.AmmInAdr	:= iAdrAmmBase2MM;
	xMsg3484.AmmOutAdr	:= iAdrMM2AmmBase;

	xMsg3485.Num 		:= 3485;
	xMsg3485.AmmInAdr	:= iAdrAmmBase2MM;
	xMsg3485.AmmOutAdr	:= iAdrMM2AmmBase;

	xMsg3486.Num 		:= 3486;
	xMsg3486.AmmInAdr	:= iAdrAmmBase2MM;
	xMsg3486.AmmOutAdr	:= iAdrMM2AmmBase;

	xMsg3487.Num 		:= 3487;
	xMsg3487.AmmInAdr	:= iAdrAmmBase2MM;
	xMsg3487.AmmOutAdr	:= iAdrMM2AmmBase;

	xMsg3488.Num 		:= 3488;
	xMsg3488.AmmInAdr	:= iAdrAmmBase2MM;
	xMsg3488.AmmOutAdr	:= iAdrMM2AmmBase;

	xMsg3489.Num 		:= 3489;
	xMsg3489.AmmInAdr	:= iAdrAmmBase2MM;
	xMsg3489.AmmOutAdr	:= iAdrMM2AmmBase;

	xMsg9077.Num 		:= 9077;
	xMsg9077.AmmInAdr	:= iAdrAmmBase2MM;
	xMsg9077.AmmOutAdr	:= iAdrMM2AmmBase;

	xMsg9079.Num 		:= 9079;
	xMsg9079.AmmInAdr	:= iAdrAmmBase2MM;
	xMsg9079.AmmOutAdr	:= iAdrMM2AmmBase;

	xMsg9080.Num 		:= 9080;
	xMsg9080.AmmInAdr	:= iAdrAmmBase2MM;
	xMsg9080.AmmOutAdr	:= iAdrMM2AmmBase;

	xMsg9081.Num 		:= 9081;
	xMsg9081.AmmInAdr	:= iAdrAmmBase2MM;
	xMsg9081.AmmOutAdr	:= iAdrMM2AmmBase;

	xMsg9082.Num 		:= 9082;
	xMsg9082.AmmInAdr	:= iAdrAmmBase2MM;
	xMsg9082.AmmOutAdr	:= iAdrMM2AmmBase;

	xMsg9201.Num 		:= 9201;
	xMsg9201.AmmInAdr	:= iAdrAmmBase2MM;
	xMsg9201.AmmOutAdr	:= iAdrMM2AmmBase;

	xMsg9202.Num 		:= 9202;
	xMsg9202.AmmInAdr	:= iAdrAmmBase2MM;
	xMsg9202.AmmOutAdr	:= iAdrMM2AmmBase;

	xMsg9203.Num 		:= 9203;
	xMsg9203.AmmInAdr	:= iAdrAmmBase2MM;
	xMsg9203.AmmOutAdr	:= iAdrMM2AmmBase;

	xMsg9204.Num 		:= 9204;
	xMsg9204.AmmInAdr	:= iAdrAmmBase2MM;
	xMsg9204.AmmOutAdr	:= iAdrMM2AmmBase;

	xMsg9205.Num 		:= 9205;
	xMsg9205.AmmInAdr	:= iAdrAmmBase2MM;
	xMsg9205.AmmOutAdr	:= iAdrMM2AmmBase;

	xMsg9206.Num 		:= 9206;
	xMsg9206.AmmInAdr	:= iAdrAmmBase2MM;
	xMsg9206.AmmOutAdr	:= iAdrMM2AmmBase;

	xMsg9207.Num 		:= 9207;
	xMsg9207.AmmInAdr	:= iAdrAmmBase2MM;
	xMsg9207.AmmOutAdr	:= iAdrMM2AmmBase;

	xMsg9208.Num 		:= 9208;
	xMsg9208.AmmInAdr	:= iAdrAmmBase2MM;
	xMsg9208.AmmOutAdr	:= iAdrMM2AmmBase;

	xMsg9209.Num 		:= 9209;
	xMsg9209.AmmInAdr	:= iAdrAmmBase2MM;
	xMsg9209.AmmOutAdr	:= iAdrMM2AmmBase;

	xMsg9210.Num 		:= 9210;
	xMsg9210.AmmInAdr	:= iAdrAmmBase2MM;
	xMsg9210.AmmOutAdr	:= iAdrMM2AmmBase;

	xMsg9211.Num 		:= 9211;
	xMsg9211.AmmInAdr	:= iAdrAmmBase2MM;
	xMsg9211.AmmOutAdr	:= iAdrMM2AmmBase;

	xMsg9212.Num 		:= 9212;
	xMsg9212.AmmInAdr	:= iAdrAmmBase2MM;
	xMsg9212.AmmOutAdr	:= iAdrMM2AmmBase;

	xMsg9233.Num 		:= 9233;
	xMsg9233.AmmInAdr	:= iAdrAmmBase2MM;
	xMsg9233.AmmOutAdr	:= iAdrMM2AmmBase;

	xMsg9234.Num 		:= 9234;
	xMsg9234.AmmInAdr	:= iAdrAmmBase2MM;
	xMsg9234.AmmOutAdr	:= iAdrMM2AmmBase;

	xMsg9235.Num 		:= 9235;
	xMsg9235.AmmInAdr	:= iAdrAmmBase2MM;
	xMsg9235.AmmOutAdr	:= iAdrMM2AmmBase;

	xMsg9236.Num 		:= 9236;
	xMsg9236.AmmInAdr	:= iAdrAmmBase2MM;
	xMsg9236.AmmOutAdr	:= iAdrMM2AmmBase;

	xMsg9250.Num 		:= 9250;
	xMsg9250.AmmInAdr	:= iAdrAmmBase2MM;
	xMsg9250.AmmOutAdr	:= iAdrMM2AmmBase;

	xMsg9251.Num 		:= 9251;
	xMsg9251.AmmInAdr	:= iAdrAmmBase2MM;
	xMsg9251.AmmOutAdr	:= iAdrMM2AmmBase;

	xMsg9252.Num 		:= 9252;
	xMsg9252.AmmInAdr	:= iAdrAmmBase2MM;
	xMsg9252.AmmOutAdr	:= iAdrMM2AmmBase;

	xMsg9277.Num 		:= 9277;
	xMsg9277.AmmInAdr	:= iAdrAmmBase2MM;
	xMsg9277.AmmOutAdr	:= iAdrMM2AmmBase;

	xMsg9278.Num 		:= 9278;
	xMsg9278.AmmInAdr	:= iAdrAmmBase2MM;
	xMsg9278.AmmOutAdr	:= iAdrMM2AmmBase;

	xMsg9379.Num 		:= 9379;
	xMsg9379.AmmInAdr	:= iAdrAmmBase2MM;
	xMsg9379.AmmOutAdr	:= iAdrMM2AmmBase;

	xMsg9380.Num 		:= 9380;
	xMsg9380.AmmInAdr	:= iAdrAmmBase2MM;
	xMsg9380.AmmOutAdr	:= iAdrMM2AmmBase;
END_PROGRAM
```

#### MsgEM.var - Local variables
```iecst
VAR
	iAdrAmmBase2MM : UDINT;
	iAdrMM2AmmBase : UDINT;
	xMsg2276 : Msg; (*NOx deviation --> canceled*)
	xMsg2446 : Msg; (*SCR BUS communication interrupted*)
	xMsg2447 : Msg; (*SCR Measuring signal failure urea pressure before dosing*)
	xMsg2448 : Msg; (*SCR Urea pressure before dosing minimum*)
	xMsg2449 : Msg; (*SCR Urea pressure before dosing maximum*)
	xMsg2450 : Msg; (*SCR Leakage in urea dosing cabinet*)
	xMsg2451 : Msg; (*SCR Urea dosing valve - error*)
	xMsg2452 : Msg; (*SCR Measuring signal failure urea flow rate after dosing*)
	xMsg2453 : Msg; (*SCR Urea flow rate - valve characteristic deviating maximum*)
	xMsg2454 : Msg; (*SCR Compressed air supply pressure urea injection maximum*)
	xMsg2455 : Msg; (*SCR Deviation to continous emission monitoring system maximum*)
	xMsg2456 : Msg; (*SCR Emission measurement line 1 - O2 maximum*)
	xMsg2457 : Msg; (*SCR Measuring signal failure emission measurement line 1 - O2 sensor*)
	xMsg2458 : Msg; (*SCR Measuring signal failure emission measurement line 2 - NO2 sensor*)
	xMsg2464 : Msg; (*SCR Urea dosing unit (external) - error*)
	xMsg2607 : Msg; (*CAN failure - NOx sensor CAN interface 1*)
	xMsg2609 : Msg; (*CAN failure - NOx sensor CAN interface 2*)
	xMsg2610 : Msg; (*No connection to the sensor - NOx sensor engine out*)
	xMsg2697 : Msg; (*SCR Urea dosing unit - maintenance needed*)
	xMsg2766 : Msg; (*Catalyst temperature minimum*)
	xMsg2769 : Msg; (*SCR Emission measurement air line - moisture maximum*)
	xMsg2877 : Msg; (*SCR Exhaust after treatment (SCR) deactivated --> canceled*)
	xMsg2878 : Msg; (*SCR Urea dosing activated*)
	xMsg2879 : Msg; (*SCR Urea dosing deactivated*)
	xMsg2884 : Msg; (*SCR Manual mode on*)
	xMsg2885 : Msg; (*SCR Manual mode off*)
	xMsg2923 : Msg; (*SCR NH3 slip detection started*)
	xMsg2924 : Msg; (*SCR NH3 slip detection completed*)
	xMsg2971 : Msg; (*Error during self-diagnosis - NOx sensor engine out*)
	xMsg2974 : Msg; (*Error during self-diagnosis - NOx sensor engine out A*)
	xMsg2977 : Msg; (*Error during self-diagnosis - NOx sensor engine out B*)
	xMsg2980 : Msg; (*Error during self-diagnosis - NOx sensor CAT out*)
	xMsg3379 : Msg; (*SCR Exhaust temperatures CAT maximum*)
	xMsg3380 : Msg; (*SCR CO emission average maximum --> canceled with V04.07*)
	xMsg3381 : Msg; (*NOx emissions - short-term average high*)
	xMsg3383 : Msg; (*SCR Measuring signal failure exhaust temperatures CAT*)
	xMsg3450 : Msg; (*SCR Group alarm - exhaust after treatment system --> canceled*)
	xMsg3451 : Msg; (*SCR Power supply to the valves interrupted*)
	xMsg3452 : Msg; (*SCR Measuring signal failure urea pressure after dosing*)
	xMsg3453 : Msg; (*SCR Urea pressure after dosing maximum*)
	xMsg3454 : Msg; (*SCR Urea pressure after dosing minimum*)
	xMsg3455 : Msg; (*SCR Urea flow rate after dosing maximum*)
	xMsg3456 : Msg; (*SCR Urea dosing pump - error*)
	xMsg3457 : Msg; (*SCR Urea-air valve blocked*)
	xMsg3458 : Msg; (*SCR Urea tank level minimum*)
	xMsg3459 : Msg; (*SCR Urea tank level minimum - dosing deactivated*)
	xMsg3460 : Msg; (*SCR Urea supply pump not operating*)
	xMsg3461 : Msg; (*SCR Measuring signal failure compressed air supply pressure urea injection*)
	xMsg3462 : Msg; (*SCR Compressed air supply pressure urea injection minimum*)
	xMsg3463 : Msg; (*SCR Compressed air valve urea injection power supply interrupted*)
	xMsg3464 : Msg; (*SCR Measuring signal failure exhaust pressure CAT inlet*)
	xMsg3465 : Msg; (*SCR Measuring signal failure exhaust pressure CAT outlet*)
	xMsg3466 : Msg; (*SCR Measuring signal failure exhaust temperature CAT inlet*)
	xMsg3467 : Msg; (*SCR Measuring signal failure exhaust temperature CAT outlet*)
	xMsg3469 : Msg; (*SCR Exhaust differential pressure CAT maximum*)
	xMsg3470 : Msg; (*SCR Emission measurement sample gas cooler - error*)
	xMsg3471 : Msg; (*SCR Emission measurement line 1 - sample gas pump not ready*)
	xMsg3472 : Msg; (*SCR Emission measurement line 2 - sample gas pump not ready*)
	xMsg3473 : Msg; (*SCR Emission measurement line 1 - moisture maximum*)
	xMsg3474 : Msg; (*SCR Emission measurement line 2 - moisture maximum*)
	xMsg3475 : Msg; (*SCR Emission measurement line 1 - flow rate minimum*)
	xMsg3476 : Msg; (*SCR Emission measurement line 2 - flow rate minimum*)
	xMsg3477 : Msg; (*SCR Measuring signal failure emission measurement line 2 - NO sensor*)
	xMsg3478 : Msg; (*SCR Measuring signal failure emission measurement line 1 - NO sensor*)
	xMsg3479 : Msg; (*SCR Measuring signal failure emission measurement line 1 - NO2 sensor*)
	xMsg3480 : Msg; (*SCR NH3 slip detection deactivated*)
	xMsg3481 : Msg; (*SCR Measuring signal failure emission measurement line 1 - CO sensor*)
	xMsg3482 : Msg; (*SCR NOx emission to check --> canceled with V04.07*)
	xMsg3483 : Msg; (*SCR CO emission to check --> canceled with V04.07*)
	xMsg3484 : Msg; (*CO emissions - short-term average high*)
	xMsg3485 : Msg; (*NOx emissions - short-term average high*)
	xMsg3486 : Msg; (*SCR Urea flow rate after dosing minimum*)
	xMsg3487 : Msg; (*SCR Exhaust temperature CAT inlet maximum*)
	xMsg3488 : Msg; (*SCR Exhaust temperature CAT outlet maximum*)
	xMsg3489 : Msg; (*SCR Emergency Stop SCR control cabinet --> canceled*)
	xMsg9077 : Msg; (*SCR NH3 slip detection interrupted*)
	xMsg9079 : Msg; (*SCR Urea dosing - dosing conditions reached*)
	xMsg9080 : Msg; (*SCR Urea dosing - dosing conditions ended*)
	xMsg9081 : Msg; (*SCR Urea dosing - requested*)
	xMsg9082 : Msg; (*SCR Urea dosing - unrequested*)
	xMsg9201 : Msg; (*Measuring signal failure O2, NOx sensor engine out*)
	xMsg9202 : Msg; (*Measuring signal failure NOx, NOx sensor engine out*)
	xMsg9203 : Msg; (*No connection to the sensor - NOx sensor engine out A*)
	xMsg9204 : Msg; (*Measuring signal failure O2, NOx sensor engine out – bank A*)
	xMsg9205 : Msg; (*Measuring signal failure NOx, NOx sensor engine out – bank A*)
	xMsg9206 : Msg; (*No connection to the sensor - NOx sensor engine out B*)
	xMsg9207 : Msg; (*Measuring signal failure O2, NOx sensor engine out – bank B*)
	xMsg9208 : Msg; (*Measuring signal failure NOx, NOx sensor engine out – bank B*)
	xMsg9209 : Msg; (*No connection to the sensor - NOx sensor CAT out*)
	xMsg9210 : Msg; (*Measuring signal failure O2, NOx sensor CAT out*)
	xMsg9211 : Msg; (*Measuring signal failure NOx, NOx sensor CAT out*)
	xMsg9212 : Msg; (*SCR Air compressor - maintenance needed *)
	xMsg9233 : Msg; (*Lifetime reached - NOx sensor engine out*)
	xMsg9234 : Msg; (*Lifetime reached - NOx sensor engine out A*)
	xMsg9235 : Msg; (*Lifetime reached - NOx sensor engine out B*)
	xMsg9236 : Msg; (*Lifetime reached - NOx sensor CAT out*)
	xMsg9250 : Msg; (*O2 deviation bank A/B maximum - NOx sensor engine out*)
	xMsg9251 : Msg; (*NOx deviation bank A/B maximum - NOx sensor engine out*)
	xMsg9252 : Msg; (*NOx emissions - daily average high*)
	xMsg9277 : Msg; (*SCR Urea dosing stopped - error*)
	xMsg9278 : Msg; (*SCR Catalyst - failure*)
	xMsg9379 : Msg; (*SCR Measuring signal failure urea tank level*)
	xMsg9380 : Msg; (*SCR Urea flow dosing error*)
	xTOF_CatOut_DiagErr : TOF; (*FuB*)
	xTOF_EngOut_A_DiagErr : TOF; (*FuB*)
	xTOF_EngOut_B_DiagErr : TOF; (*FuB*)
	xTOF_EngOut_DiagErr : TOF; (*FuB*)
	xTON_T_SCR_Cat3 : TON := (0); (*FuB*)
END_VAR
```

### Program Logical/Emission/ParEM (IEC, version 4.06.0) - + parameter storage and modulstate communication

- perm_par.st (not readable text: treated as protected, skipped)

#### perm_par.var
```iecst
VAR
	tParaIntern : ParaHandler_typ; (*Connector type to perm_par*)
	tMM2ParaBase_ReadBack : MM2ParaBase_type; (*INTERNAL! V4.06 new readback structure for information from previous tasks*)
	bWriteDataObj : BOOL; (* TRUE=write data object module *)
	bDataObjLenErr : BOOL; (*Error occured in permem: data module size missmatch*)
	bCreateDataObj : BOOL; (* TRUE=create new data object *)
	bWriteOnce : BOOL; (* write permanent memory once *)
	DatObjCreate_01 : DatObjCreate; (* data object create *)
	DatObjInfoBak_02 : DatObjInfo; (* data object info *)
	DatObjDelete_01 : DatObjDelete; (* data object delete *)
	DatObjRead_01 : DatObjRead; (* data object read *)
	DatObjRead_02 : DatObjRead; (* manual initiated data object read *)
	DatObjWrite_01 : DatObjWrite; (* data object write *)
	DatObjDelete_02 : DatObjDelete; (* data object delete *)
	DatObjDelete_11 : DatObjDelete; (*Delete Backup File*)
	DatObjInfo_01 : DatObjInfo; (* data object info *)
	DatObjInfo_02 : DatObjInfo; (* data object info *)
	szModuleName : STRING[35]; (* module name of object *)
	szModuleNameBackup : STRING[35]; (* module name of posiibly created backup object *)
	DatObjCopy_01 : DatObjCopy;
	bCopyDataObj : BOOL;
	TON_WarnDelay : TON;
	TON_WritePMEM : TON; (* delay write permanent memory *)
	ulPMPointer : UDINT; (* adress of actual checksum value *)
	ulChecksum : UDINT; (* parameter checksum value *)
	pm_len : UDINT; (* permanent value lenght *)
	ulChecksumOld : UDINT; (* last vlaue of parameter checksum *)
	ulChkValue : UDINT; (* actual value of parameter pointer *)
	pm_id : UDINT; (* permanent value identifier *)
	pm_p : UDINT; (* permanent value pointer *)
	DatObjInfo_META : DatObjInfo;
	DatObjRead_META : DatObjRead;
	szMetaDataRaw : STRING[2000];
	szMetaData : ARRAY[0..4] OF STRING[35];
	szMetaDataVis : ARRAY[0..3] OF STRING[35];
	ssIndex : INT;
	ssCount : INT;
	ucMetaDataRaw : ARRAY[0..2000] OF USINT;
	ssCount2 : INT;
	szMetaDataFile : STRING[10];
	szText1 : STRING[20];
	pv_adr_IN_XX_tPB2MM : UDINT;
	pv_lng : UDINT;
	pv_lng_IN_XX_tPB2MM : UDINT;
	pv_lng_OUT_XX_tPB2MM : UDINT;
	szText2 : STRING[20];
	pv_adr_OUT_XX_tXX2PB : UDINT;
END_VAR
VAR CONSTANT
	ERR_NOERROR : UINT := 0;
END_VAR
VAR
	usPMWriteCnt : UINT;
	pm_Error : UDINT; (* permanent value error *) (* Deleted: pm : ParaMem_typ; permanent memory tags mathias, 22.8.11*)
	fun_Error : UDINT := 0; (*state > 0 = function error*)
	xLocalParaCheck : ParaCheckFUB; (*local function instance to check parameter values*)
	TON_ParaSetupOk : TON;
	bParaCheckSystemOk : BOOL;
	iDebug_ParaOkChecked : UDINT;
	bRestoreBackupDataObj : BOOL := FALSE;
	bRestoreDataObjContent : BOOL := FALSE;
	pm_id_backup : UDINT;
	pm_p_Backup : UDINT;
	DatObjCopy_02 : DatObjCopy;
	bDeleteBackupDataObj : BOOL := FALSE; (*Command to delete backup data module file on purpose*)
	bDebugPara : ARRAY[0..5] OF BOOL;
	ssIndex2 : INT;
	ssIndex3 : INT;
	ssIndex4 : INT;
	ssIndexVis : INT;
	szText : STRING[40];
	pv_adr_Para : UDINT;
	szParaSnippet : ARRAY[0..5] OF STRING[150];
	szParaIndex : STRING[10];
	slValue : DINT;
	iModuleDLD_ResetCount : INT;
	bDownloadDetected : BOOL;
	bFlagParaStructCopyWorking : BOOL; (*true, if cyclic para copying is active, 1 false cycle at every copy *)
	bStoreInitParaInDataObj : BOOL := FALSE;
	bTestflag : BOOL;
	bReadOutMETA_Once : BOOL;
	tParaCheck_iPvAdress : ARRAY[0..5] OF UDINT;
	tParaCheck_iPvLengt : ARRAY[0..5] OF UDINT;
	tParaCheck_rPvValue : ARRAY[0..5] OF REAL;
	tParaCheck_rRangeMIN : ARRAY[0..5] OF REAL;
	tParaCheck_rRangeMAX : ARRAY[0..5] OF REAL;
	tParaCheck_szPvName : ARRAY[0..5] OF STRING[35];
	ssFormatDetected : INT;
	szMetaDataPart : STRING[150];
	szFullTaskName : STRING[35];
	szFullMetaModuleName : STRING[35];
	debugLen : INT;
	debugSize : INT := 0;
	strcat_adr1 : UDINT;
	strcat_adr2 : UDINT;
	ssIndexTN : INT;
	bAlternate : BOOL;
	n : INT;
	iAlternateChecksum : DINT;
	iAlternateChecksumOld : DINT;
	ulDebugChkValue : ARRAY[0..999] OF UDINT;
	Adr1 : UDINT;
	Adr2 : UDINT;
	usPMWriteCntStepsize : UINT := 1; (*different step sizes to help debug*)
	usPMWriteCntXOR : UINT;
	usPMWriteCntAltSum : UINT;
	ulAdrPM : UDINT;
	usChkValuePM : USINT;
	ulAdrPara : UDINT;
	ulPara_len : UDINT;
	usChkValuePara : USINT;
	iDebugCountPMDifferences : DINT := 0;
	bEngineRunDetected : BOOL; (*detection status bit autocommand 100 /101  for engine run state*)
	ucMetaDataDebugInfoLine : ARRAY[0..24] OF STRING[80];
	ssIndexMand : INT := 0;
	szMetaDataMand : STRING[35];
	iMyErrorInfo_Autoreset : DINT; (*internal autoreset counter*)
	ssIndex_Version : INT; (*internal*)
	ssIndex_BU : INT; (*internal*)
	ssIndex_BU2 : INT; (*internal*)
END_VAR
```

### Program Logical/Emission/PermEM (IEC, version 4.10.0) - + PermanentMemory

- PermEMCyclic.st (not readable text: treated as protected, skipped)

- PermEMInit.st (not readable text: treated as protected, skipped)

#### PermEM.var
```iecst
VAR
	bCreateDataObj : BOOL;
	bWriteDataObj : BOOL;
	DatObjCreate_01 : DatObjCreate;
	DatObjDelete_PermMem : DatObjDelete;
	DatObjInfo_01 : DatObjInfo;
	DatObjRead_01 : DatObjRead;
	DatObjWrite_01 : DatObjWrite;
END_VAR
VAR CONSTANT
	ERR_NOERROR : UINT := 0;
END_VAR
VAR
	ModulName : STRING[35];
	perm_par_vers : UINT;
	pmm : Perm_EM_Struct;
	pm_Error : UINT;
	pm_id : UDINT;
	pm_len : UDINT;
	pm_p : UDINT;
	TON_WritePMEM : TON;
	ulChecksum : UDINT;
	ulChecksumOld : UDINT;
	ulChkValue : UDINT;
	ulPMPointer : UDINT;
	write_once : BOOL;
	TON_WarnDelay : TON;
	TON_BlockMinFileAge : TON; (*waiting time without file write after successful performed write*)
	bBlock_MinFileAge : BOOL := FALSE; (*pause the perm file write after each sucessful write*)
	iPM_WriteCnt : UDINT; (* *) (*old VarName: usPMWriteCnt*)
END_VAR
```

### Package Logical/EngineController - EC: Engine Controller

### Library Logical/EngineController/Lib_EC/lSimPIDx (ANSIC)

#### lSimPIDx.fun
```iecst
FUNCTION_BLOCK fSimPIDx
  VAR_INPUT
    ssMethodType: SINT;
  END_VAR  VAR_INPUT
        P : REAL; (*Proportional Gain*)
  END_VAR
  VAR_INPUT
        I : REAL; (*Integral Gain*)
  END_VAR
  VAR_INPUT
        D : REAL; (*Differential Gain*)
  END_VAR
  VAR_INPUT
        N : REAL; (*Filter Coefficient*)
  END_VAR
  VAR_INPUT
        wxmax : LREAL; (*Maximum Input*)
  END_VAR
  VAR_INPUT
        wxmin : LREAL; (*Minimum Input*)
  END_VAR
  VAR_INPUT
        umax : REAL; (*Upper Output Saturation Level*)
  END_VAR
  VAR_INPUT
        umin : REAL; (*Lower Output Saturation Level*)
  END_VAR
  VAR_INPUT
        Kt : REAL; (*Tracking Gain*)
  END_VAR
  VAR_INPUT
        deadband : LREAL; (*Deadband*)
  END_VAR
  VAR_INPUT
        mode : USINT; (*Mode*)
  END_VAR
  VAR_INPUT
        u_man : REAL; (*Manual Value*)
  END_VAR
  VAR_INPUT
        a : REAL; (*Feedforward Value*)
  END_VAR
  VAR_INPUT
        invert : BOOL := FALSE; (*Invert*)
  END_VAR
  VAR_INPUT
        w : REAL; (*Reference Value*)
  END_VAR
  VAR_INPUT
        x : REAL; (*Actual Value*)
  END_VAR
  VAR_INPUT
        reset : BOOL := FALSE; (*Reset*)
  END_VAR
  VAR_INPUT
        I0 : REAL; (*I Integrator Reset*)
  END_VAR
  VAR_INPUT
        D0 : REAL; (*D Integrator Reset (Filter)*)
  END_VAR
  VAR_OUTPUT
        u : REAL; (*Controller Output*)
  END_VAR
  VAR_OUTPUT
        up : REAL; (*Proportional Output*)
  END_VAR
  VAR_OUTPUT
        ui : REAL; (*Integral Output*)
  END_VAR
  VAR_OUTPUT
        ud : REAL; (*Differential Output*)
  END_VAR
  VAR_OUTPUT
        u_tr : REAL; (*Tracking Output*)
  END_VAR
  VAR_INPUT
        e_int : REAL; (*external input for integral control*)
  END_VAR
  VAR_INPUT
        fbk_mode : USINT; (*Anti Windup Feedback Mode*)
  END_VAR
  VAR_INPUT
        u_fbk : REAL; (*External Anti Windup Feedback Value*)
  END_VAR
	VAR
		bur_BlockIO_SimPIDBR6 : BlockIO_SimPIDBR6;
	END_VAR
	VAR
		bur_D_Work_SimPIDBR6 : D_Work_SimPIDBR6;
	END_VAR
END_FUNCTION_BLOCK
```

#### lSimPIDx.typ
```iecst
TYPE

END_TYPE
TYPE
BlockIO_SimPIDBR6 : STRUCT
	Input10 : REAL;
	Input6 : REAL;
	Input4 : REAL;
	Input : REAL;
	Gain : REAL;
	Input2 : REAL;
	Integrator : REAL;
	Input3 : REAL;
	FilterCoefficient : REAL;
	Saturation : REAL;
	Modeswitch : REAL;
	Input11 : REAL;
	Input8 : REAL;
	Input9 : USINT;
	Input7 : USINT;
	Input5 : BOOL;
	Input1 : BOOL;
END_STRUCT;
D_Work_SimPIDBR6 : STRUCT
	Integrator_DSTATE : REAL;
	Filter_DSTATE : REAL;
	Integrator_IC_LOADING : USINT;
	Filter_IC_LOADING : USINT;
END_STRUCT;
END_TYPE
```

#### SimPIDBR6.h
```c
/********************************************************************
 * COPYRIGHT -- Bernecker + Rainer Industrie-Elektronik Ges.m.b.H.
 ********************************************************************
 * Program: SimPIDBR6
 * File: SimPIDBR6.h
 * Author: 105055527
 * Created: Tue Dec 06 16:11:54 2016
 ********************************************************************
 * Header for program SimPIDBR6
 ********************************************************************
 * Generated with B&R Automation Studio Target for Simulink V4.2
 * (ERT based)
 ********************************************************************/

#ifndef RTW_HEADER_SimPIDBR6_h_
#define RTW_HEADER_SimPIDBR6_h_
#ifndef SimPIDBR6_COMMON_INCLUDES_
# define SimPIDBR6_COMMON_INCLUDES_
#include <math.h>
#include "rtwtypes.h"
#endif                                 /* SimPIDBR6_COMMON_INCLUDES_ */

#include "SimPIDBR6_types.h"
#include "lSimPIDx.h"

/* Macros for accessing real-time model data structure */
#ifndef rtmGetErrorStatus
# define rtmGetErrorStatus(rtm)        ((void*) 0)
#endif

#ifndef rtmSetErrorStatus
# define rtmSetErrorStatus(rtm, val)   ((void) 0)
#endif

#ifndef rtmGetStopRequested
# define rtmGetStopRequested(rtm)      ((void*) 0)
#endif

#ifndef MIN
#define MIN(a,b)                       ((a) < (b) ? (a) : (b))
#endif

#ifndef MAX
#define MAX(a,b)                       ((a) > (b) ? (a) : (b))
#endif

/* Block signals (auto storage) */

/* Block states (auto storage) for system '<Root>' */

/* Model entry point functions */
extern void SimPIDBR6_initialize(D_Work_SimPIDBR6 *SimPIDBR6_DWork, struct fSimPIDx* inst);
extern void SimPIDBR6_step(BlockIO_SimPIDBR6 *SimPIDBR6_B, D_Work_SimPIDBR6
  *SimPIDBR6_DWork, struct fSimPIDx* inst);
extern void SimPIDBR6_terminate(struct fSimPIDx* inst);

/*-
 * The generated code includes comments that allow you to trace directly
 * back to the appropriate location in the model.  The basic format
 * is <system>/block_name, where system is the system number (uniquely
 * assigned by Simulink) and block_name is the name of the block.
 *
 * Use the MATLAB hilite_system command to trace the generated code back
 * to the model.  For example,
 *
 * hilite_system('<S3>')    - opens system 3
 * hilite_system('<S3>/Kp') - opens and selects block Kp which resides in S3
 *
 * Here is the system hierarchy for this model
 *
 * '<Root>' : 'SimPIDBR6'
 * '<S1>'   : 'SimPIDBR6/PID Autocoding'
 * '<S2>'   : 'SimPIDBR6/PID Autocoding/PID'
 * '<S3>'   : 'SimPIDBR6/PID Autocoding/PID/Clamping circuit'
 * '<S4>'   : 'SimPIDBR6/PID Autocoding/PID/Clamping circuit/Compare To Constant'
 */
#endif                                 /* RTW_HEADER_SimPIDBR6_h_ */
```

#### SimPIDBR6_private.h
```c
/********************************************************************
 * COPYRIGHT -- Bernecker + Rainer Industrie-Elektronik Ges.m.b.H.
 ********************************************************************
 * Program: SimPIDBR6
 * File: SimPIDBR6_private.h
 * Author: 105055527
 * Created: Tue Dec 06 16:11:54 2016
 ********************************************************************
 * Header for program SimPIDBR6
 ********************************************************************
 * Generated with B&R Automation Studio Target for Simulink V4.2
 * (ERT based)
 ********************************************************************/

#ifndef RTW_HEADER_SimPIDBR6_private_h_
#define RTW_HEADER_SimPIDBR6_private_h_
#include "rtwtypes.h"
#include <bur/plctypes.h>
#ifndef __RTWTYPES_H__
#error This file requires rtwtypes.h to be included
#else
#ifdef TMWTYPES_PREVIOUSLY_INCLUDED
#error This file requires rtwtypes.h to be included before tmwtypes.h
#else

/* Check for inclusion of an incorrect version of rtwtypes.h */
#ifndef RTWTYPES_ID_C08S16I32L32N32F1
#error This code was generated with a different "rtwtypes.h" than the file included
#endif                                 /* RTWTYPES_ID_C08S16I32L32N32F1 */
#endif                                 /* TMWTYPES_PREVIOUSLY_INCLUDED */
#endif                                 /* __RTWTYPES_H__ */

#ifndef MIN
#define MIN(a,b)                       ((a) < (b) ? (a) : (b))
#endif

#ifndef MAX
#define MAX(a,b)                       ((a) > (b) ? (a) : (b))
#endif

/* Imported (extern) block parameters */
extern real_T deadband;                /* Variable: deadband
                                        * Referenced by: '<S1>/Deadband'
                                        */
extern real_T wxmax;                   /* Variable: wxmax
                                        * Referenced by: '<S1>/Scaling'
                                        */
extern real_T wxmin;                   /* Variable: wxmin
                                        * Referenced by: '<S1>/Scaling'
                                        */
extern real32_T D;                     /* Variable: D
                                        * Referenced by: '<S2>/Gain2'
                                        */
extern real32_T I;                     /* Variable: I
                                        * Referenced by: '<S2>/Gain1'
                                        */
extern real32_T Kt;                    /* Variable: Kt
                                        * Referenced by: '<S1>/Constant'
                                        */
extern real32_T N;                     /* Variable: N
                                        * Referenced by: '<S2>/Filter Coefficient'
                                        */
extern real32_T P;                     /* Variable: P
                                        * Referenced by: '<S2>/Gain'
                                        */
extern real32_T umax;                  /* Variable: umax
                                        * Referenced by: '<S2>/Saturation'
                                        */
extern real32_T umin;                  /* Variable: umin
                                        * Referenced by: '<S2>/Saturation'
                                        */

#endif                                 /* RTW_HEADER_SimPIDBR6_private_h_ */
```

#### SimPIDBR6_types.h
```c
/********************************************************************
 * COPYRIGHT -- Bernecker + Rainer Industrie-Elektronik Ges.m.b.H.
 ********************************************************************
 * Program: SimPIDBR6
 * File: SimPIDBR6_types.h
 * Author: 105055527
 * Created: Tue Dec 06 16:11:54 2016
 ********************************************************************
 * Header for program SimPIDBR6
 ********************************************************************
 * Generated with B&R Automation Studio Target for Simulink V4.2
 * (ERT based)
 ********************************************************************/

#ifndef RTW_HEADER_SimPIDBR6_types_h_
#define RTW_HEADER_SimPIDBR6_types_h_
#ifndef MIN
#define MIN(a,b)                       ((a) < (b) ? (a) : (b))
#endif

#ifndef MAX
#define MAX(a,b)                       ((a) > (b) ? (a) : (b))
#endif
#endif                                 /* RTW_HEADER_SimPIDBR6_types_h_ */
```

#### rtwtypes.h
```c
/********************************************************************
 * COPYRIGHT -- Bernecker + Rainer Industrie-Elektronik Ges.m.b.H.
 ********************************************************************
 * Program: SimPIDBR6
 * File: rtwtypes.h
 * Author: 105055527
 * Created: Tue Dec 06 16:11:54 2016
 ********************************************************************
 * Header for program SimPIDBR6
 ********************************************************************
 * Generated with B&R Automation Studio Target for Simulink V4.2
 * (ERT based)
 ********************************************************************/

#ifndef __RTWTYPES_H__
#define __RTWTYPES_H__
#ifndef TRUE
# define TRUE                          (1U)
#endif

#ifndef FALSE
# define FALSE                         (0U)
#endif

#ifndef __TMWTYPES__
#define __TMWTYPES__
#include <limits.h>

/*=======================================================================*
 * Target hardware information
 *   Device type: Intel->x86/Pentium
 *   Number of bits:     char:   8    short:   16    long:  32
 *                       long:  32
 *                       native word size:  32
 *   Byte ordering: LittleEndian
 *   Signed integer division rounds to: Zero
 *   Shift right on a signed integer as arithmetic shift: on
 *=======================================================================*/

/*=======================================================================*
 * Fixed width word size data types:                                     *
 *   int8_T, int16_T, int32_T     - signed 8, 16, or 32 bit integers     *
 *   uint8_T, uint16_T, uint32_T  - unsigned 8, 16, or 32 bit integers   *
 *   real32_T, real64_T           - 32 and 64 bit floating point numbers *
 *=======================================================================*/
typedef signed char int8_T;
typedef unsigned char uint8_T;
typedef short int16_T;
typedef unsigned short uint16_T;
typedef long int32_T;
typedef unsigned long uint32_T;
typedef float real32_T;
typedef double real64_T;

/*===========================================================================*
 * Generic type definitions: real_T, time_T, boolean_T, int_T, uint_T,       *
 *                           ulong_T, char_T and byte_T.                     *
 *===========================================================================*/
typedef double real_T;
typedef double time_T;
typedef unsigned char boolean_T;
typedef long int_T;
typedef unsigned long uint_T;
typedef unsigned long ulong_T;
typedef char char_T;
typedef unsigned char uchar_T;
typedef char_T byte_T;

/*=======================================================================*
 * Min and Max:                                                          *
 *   int8_T, int16_T, int32_T     - signed 8, 16, or 32 bit integers     *
 *   uint8_T, uint16_T, uint32_T  - unsigned 8, 16, or 32 bit integers   *
 *=======================================================================*/
#define MAX_int8_T                     ((int8_T)(127))
#define MIN_int8_T                     ((int8_T)(-128))
#define MAX_uint8_T                    ((uint8_T)(255U))
#define MIN_uint8_T                    ((uint8_T)(0U))
#define MAX_int16_T                    ((int16_T)(32767))
#define MIN_int16_T                    ((int16_T)(-32768))
#define MAX_uint16_T                   ((uint16_T)(65535U))
#define MIN_uint16_T                   ((uint16_T)(0U))
#define MAX_int32_T                    ((int32_T)(2147483647))
#define MIN_int32_T                    ((int32_T)(-2147483647-1))
#define MAX_uint32_T                   ((uint32_T)(0xFFFFFFFFU))
#define MIN_uint32_T                   ((uint32_T)(0U))

/* Logical type definitions */
#if (!defined(__cplusplus)) && (!defined(__true_false_are_keywords))
#  ifndef false
#   define false                       (0U)
#  endif

#  ifndef true
#   define true                        (1U)
#  endif
#endif

/*
 * Simulink Coder assumes the code is compiled on a target using a 2's complement representation
 * for signed integer values.
 */
#if ((SCHAR_MIN + 1) != -SCHAR_MAX)
#error "This code must be compiled using a 2's complement representation for signed integer values"
#endif

/* This ID is used to detect inclusion of an incompatible rtwtypes.h */
#define RTWTYPES_ID_C08S16I32L32N32F1
#else                                  /* __TMWTYPES__ */
#define TMWTYPES_PREVIOUSLY_INCLUDED
#endif                                 /* __TMWTYPES__ */

/* Block D-Work pointer type */
typedef void * pointer_T;

/* Simulink specific types */
#ifndef __SIMSTRUC_TYPES_H__
#define __SIMSTRUC_TYPES_H__

/* Trigger directions: falling, either, and rising */
typedef enum {
  FALLING_ZERO_CROSSING = -1,
  ANY_ZERO_CROSSING = 0,
  RISING_ZERO_CROSSING = 1
} ZCDirection;

/* Previous state of a trigger signal */
typedef uint8_T ZCSigState;

/* Initial value of a trigger zero crossing signal */
#define UNINITIALIZED_ZCSIG            0x03U
#define NEG_ZCSIG                      0x02U
#define POS_ZCSIG                      0x01U
#define ZERO_ZCSIG                     0x00U

/* Current state of a trigger signal */
typedef enum {
  FALLING_ZCEVENT = -1,
  NO_ZCEVENT = 0,
  RISING_ZCEVENT = 1
} ZCEventType;

#endif                                 /* __SIMSTRUC_TYPES_H__ */
#endif                                 /* __RTWTYPES_H__ */

#ifndef MIN
#define MIN(a,b)                       ((a) < (b) ? (a) : (b))
#endif

#ifndef MAX
#define MAX(a,b)                       ((a) > (b) ? (a) : (b))
#endif
```

#### SimPIDBR6.c
```c
/********************************************************************
 * COPYRIGHT -- Bernecker + Rainer Industrie-Elektronik Ges.m.b.H.
 ********************************************************************
 * Program: SimPIDBR6
 * File: SimPIDBR6.c
 * Author: 105055527
 * Created: Tue Dec 06 16:11:54 2016
 ********************************************************************
 * Implementation of program SimPIDBR6
 ********************************************************************
 * Generated with B&R Automation Studio Target for Simulink V4.2
 * (ERT based)
 ********************************************************************/
#include "SimPIDBR6.h"
#include "SimPIDBR6_private.h"

/*  Defines */

/*  Data Types */

/**************************** GLOBAL DATA *************************************/
/*  Definitions */

/*  Declarations  */

/***************************** FILE SCOPE DATA ********************************/

/*************************** FUNCTIONS ****************************************/

/* Model step function */
void SimPIDBR6_step(struct BlockIO_SimPIDBR6 *SimPIDBR6_B, struct D_Work_SimPIDBR6
                    *SimPIDBR6_DWork, struct fSimPIDx* inst)
{
  real_T rtb_Product;
  real_T rtb_Invertswitch;
  real32_T rtb_Product2;
  real32_T rtb_Gain2;
  real32_T rtb_Gain;
  real32_T rtb_SumI;

  /* S-Function (bur_in): '<Root>/Input9' */
  SimPIDBR6_B->Input9 = inst->mode;

  /* S-Function (bur_in): '<Root>/Input10' */
  SimPIDBR6_B->Input10 = inst->u_man;

  /* S-Function (bur_in): '<Root>/Input6' */
  SimPIDBR6_B->Input6 = inst->a;

  /* S-Function (bur_in): '<Root>/Input5' */
  SimPIDBR6_B->Input5 = inst->invert;

  /* Switch: '<S1>/Invert switch' incorporates:
   *  Constant: '<S1>/Constant2'
   *  Constant: '<S1>/Constant3'
   */
  if (SimPIDBR6_B->Input5) {
    rtb_Invertswitch = -1.0;
  } else {
    rtb_Invertswitch = 1.0;
  }

  /* End of Switch: '<S1>/Invert switch' */

  /* S-Function (bur_in): '<Root>/Input4' */
  SimPIDBR6_B->Input4 = inst->w;

  /* Product: '<S1>/Product' incorporates:
   *  Constant: '<S1>/Scaling'
   */
  rtb_Product = 1.0 / (inst->wxmax - inst->wxmin) * (real_T)SimPIDBR6_B->Input4;

  /* S-Function (bur_in): '<Root>/Input' */
  SimPIDBR6_B->Input = inst->x;

  /* Sum: '<S1>/Sum' incorporates:
   *  Constant: '<S1>/Scaling'
   *  Product: '<S1>/Product1'
   */
  rtb_Product -= 1.0 / (inst->wxmax - inst->wxmin) * (real_T)SimPIDBR6_B->Input;

  /* DeadZone: '<S1>/Deadband' */
  if (rtb_Product > inst->deadband) {
    rtb_Product -= inst->deadband;
  } else if (rtb_Product >= -inst->deadband) {
    rtb_Product = 0.0;
  } else {
    rtb_Product -= -inst->deadband;
  }

  /* End of DeadZone: '<S1>/Deadband' */

  /* Product: '<S1>/Product2' */
  rtb_Product2 = (real32_T)(rtb_Invertswitch * rtb_Product);

  /* Gain: '<S2>/Gain' */
  SimPIDBR6_B->Gain = inst->P * rtb_Product2;

  /* S-Function (bur_in): '<Root>/Input1' */
  SimPIDBR6_B->Input1 = inst->reset;

  /* S-Function (bur_in): '<Root>/Input2' */
  SimPIDBR6_B->Input2 = inst->I0;

  /* DiscreteIntegrator: '<S2>/Integrator' */
  if (SimPIDBR6_DWork->Integrator_IC_LOADING != 0) {
    SimPIDBR6_DWork->Integrator_DSTATE = SimPIDBR6_B->Input2;
  }

  if (SimPIDBR6_B->Input1) {
    SimPIDBR6_DWork->Integrator_DSTATE = SimPIDBR6_B->Input2;
  }

  SimPIDBR6_B->Integrator = SimPIDBR6_DWork->Integrator_DSTATE;

  /* End of DiscreteIntegrator: '<S2>/Integrator' */

  /* Gain: '<S2>/Gain2' */
  rtb_Gain2 = inst->D * rtb_Product2;

  /* S-Function (bur_in): '<Root>/Input3' */
  SimPIDBR6_B->Input3 = inst->D0;

  /* DiscreteIntegrator: '<S2>/Filter' */
  if (SimPIDBR6_DWork->Filter_IC_LOADING != 0) {
    SimPIDBR6_DWork->Filter_DSTATE = SimPIDBR6_B->Input3;
  }

  if (SimPIDBR6_B->Input1) {
    SimPIDBR6_DWork->Filter_DSTATE = SimPIDBR6_B->Input3;
  }

  /* Gain: '<S2>/Filter Coefficient' incorporates:
   *  DiscreteIntegrator: '<S2>/Filter'
   *  Sum: '<S2>/SumD'
   */
  SimPIDBR6_B->FilterCoefficient = (rtb_Gain2 - SimPIDBR6_DWork->Filter_DSTATE) *
    inst->N;

  /* Sum: '<S2>/Sum2' incorporates:
   *  Sum: '<S2>/Sum1'
   */
  rtb_Gain2 = ((SimPIDBR6_B->Gain + SimPIDBR6_B->Integrator) +
               SimPIDBR6_B->FilterCoefficient) + SimPIDBR6_B->Input6;

  /* Saturate: '<S2>/Saturation' */
  if (rtb_Gain2 >= inst->umax) {
    SimPIDBR6_B->Saturation = inst->umax;
  } else if (rtb_Gain2 <= inst->umin) {
    SimPIDBR6_B->Saturation = inst->umin;
  } else {
    SimPIDBR6_B->Saturation = rtb_Gain2;
  }

  /* End of Saturate: '<S2>/Saturation' */

  /* MultiPortSwitch: '<S1>/Mode switch' */
  switch (SimPIDBR6_B->Input9) {
   case 1:
    SimPIDBR6_B->Modeswitch = SimPIDBR6_B->Input10;
    break;

   case 2:
    SimPIDBR6_B->Modeswitch = SimPIDBR6_B->Input10;
    break;

   default:
    SimPIDBR6_B->Modeswitch = SimPIDBR6_B->Saturation;
    break;
  }

  /* End of MultiPortSwitch: '<S1>/Mode switch' */

  /* S-Function (bur_out): '<Root>/Output' */
  inst->u = SimPIDBR6_B->Modeswitch;

  /* S-Function (bur_out): '<Root>/Output1' */
  inst->up = SimPIDBR6_B->Gain;

  /* S-Function (bur_out): '<Root>/Output2' */
  inst->ui = SimPIDBR6_B->Integrator;

  /* S-Function (bur_out): '<Root>/Output3' */
  inst->ud = SimPIDBR6_B->FilterCoefficient;

  /* S-Function (bur_out): '<Root>/Output4' */
  inst->u_tr = SimPIDBR6_B->Saturation;

  /* S-Function (bur_in): '<Root>/Input11' */
  SimPIDBR6_B->Input11 = inst->e_int;

  /* S-Function (bur_in): '<Root>/Input7' */
  SimPIDBR6_B->Input7 = inst->fbk_mode;

  /* S-Function (bur_in): '<Root>/Input8' */
  SimPIDBR6_B->Input8 = inst->u_fbk;

  /* MultiPortSwitch: '<S2>/Multiport Switch' */
  if (SimPIDBR6_B->Input7 == 1) {
    rtb_Gain = SimPIDBR6_B->Input8;
  } else {
    rtb_Gain = SimPIDBR6_B->Saturation;
  }

  /* End of MultiPortSwitch: '<S2>/Multiport Switch' */

  /* Sum: '<S3>/Sum' */
  rtb_Gain2 = rtb_Gain - rtb_Gain2;

  /* MultiPortSwitch: '<S1>/Tracking switch' incorporates:
   *  Constant: '<S1>/Constant'
   *  Constant: '<S1>/Constant1'
   */
  switch (SimPIDBR6_B->Input9) {
   case 1:
    rtb_Invertswitch = 0.0;
    break;

   case 2:
    rtb_Invertswitch = inst->Kt;
    break;

   default:
    rtb_Invertswitch = 0.0;
    break;
  }

  /* End of MultiPortSwitch: '<S1>/Tracking switch' */

  /* Sum: '<S2>/SumI1' incorporates:
   *  Gain: '<S2>/Gain1'
   *  Product: '<S2>/Product'
   *  Sum: '<S2>/SumI3'
   */
  rtb_Product2 = (inst->I * rtb_Product2 + SimPIDBR6_B->Input11) + (real32_T)((real_T)
    (SimPIDBR6_B->Input10 - SimPIDBR6_B->Saturation) * rtb_Invertswitch);

  /* Signum: '<S3>/SignPreSat' */
  if (rtb_Gain2 < 0.0F) {
    rtb_Gain = -1.0F;
  } else if (rtb_Gain2 > 0.0F) {
    rtb_Gain = 1.0F;
  } else {
    rtb_Gain = rtb_Gain2;
  }

  /* Signum: '<S3>/SignPreIntegrator' */
  if (rtb_Product2 < 0.0F) {
    rtb_SumI = -1.0F;
  } else if (rtb_Product2 > 0.0F) {
    rtb_SumI = 1.0F;
  } else {
    rtb_SumI = rtb_Product2;
  }

  /* Switch: '<S2>/Switch' incorporates:
   *  Abs: '<S3>/Abs'
   *  Constant: '<S2>/Constant4'
   *  Constant: '<S4>/Constant'
   *  Logic: '<S3>/AND'
   *  RelationalOperator: '<S3>/Equal'
   *  RelationalOperator: '<S4>/Compare'
   *  Signum: '<S3>/SignPreIntegrator'
   *  Signum: '<S3>/SignPreSat'
   */
  if (((real32_T)fabs(rtb_Gain2) > 0.005F) && (rtb_Gain != rtb_SumI)) {
    rtb_Gain2 = 0.0F;
  } else {
    rtb_Gain2 = rtb_Product2;
  }

  /* End of Switch: '<S2>/Switch' */

  /* Update for DiscreteIntegrator: '<S2>/Integrator' */
  SimPIDBR6_DWork->Integrator_IC_LOADING = 0U;
  SimPIDBR6_DWork->Integrator_DSTATE += 0.01F * rtb_Gain2;

  /* Update for DiscreteIntegrator: '<S2>/Filter' */
  SimPIDBR6_DWork->Filter_IC_LOADING = 0U;
  SimPIDBR6_DWork->Filter_DSTATE += 0.01F * SimPIDBR6_B->FilterCoefficient;
}

/* Model initialize function */
void SimPIDBR6_initialize(struct D_Work_SimPIDBR6 *SimPIDBR6_DWork, struct fSimPIDx* inst)
{
  /* InitializeConditions for DiscreteIntegrator: '<S2>/Integrator' */
  SimPIDBR6_DWork->Integrator_IC_LOADING = 1U;

  /* InitializeConditions for DiscreteIntegrator: '<S2>/Filter' */
  SimPIDBR6_DWork->Filter_IC_LOADING = 1U;
}

/* Model terminate function */
void SimPIDBR6_terminate(struct fSimPIDx* inst)
{
  /* (no terminate code required) */
}

/*======================== TOOL VERSION INFORMATION ==========================*
 * MATLAB 8.0 (R2012b)20-Jul-2012                                             *
 * Simulink 8.0 (R2012b)20-Jul-2012                                           *
 * Simulink Coder 8.3 (R2012b)20-Jul-2012                                     *
 * Embedded Coder 6.3 (R2012b)20-Jul-2012                                     *
 * Stateflow 8.0 (R2012b)20-Jul-2012                                          *
 *============================================================================*/

/*======================= LICENSE IN USE INFORMATION =========================*
 * curve_fitting_toolbox                                                      *
 * matlab                                                                     *
 * matlab_coder                                                               *
 * real-time_workshop                                                         *
 * rtw_embedded_coder                                                         *
 * simulink                                                                   *
 *============================================================================*/
```

#### fSimPIDx.c
```c
/********************************************************************
 * COPYRIGHT -- Bernecker + Rainer Industrie-Elektronik Ges.m.b.H.
 ********************************************************************
 * Program: SimPIDBR6
 * File: fSimPIDx.c
 * Author: 105055527
 * Created: Tue Dec 06 16:11:54 2016
 ********************************************************************
 * Implementation of program SimPIDBR6
 ********************************************************************
 * Generated with B&R Automation Studio Target for Simulink V4.2
 * (ERT based)
 ********************************************************************/
#include <bur/plctypes.h>
#include "SimPIDBR6.h"
#include "rtwtypes.h"

/* Defines */
#define SS_TERMINATE 4
#define SS_OUTPUT 3
#define SS_INITIALIZE 2

/*  Data Types */

/**************************** GLOBAL DATA *************************************/
/*  Definitions */

/*  Declarations  */

/***************************** FILE SCOPE DATA ********************************/

/*************************** FUNCTIONS ****************************************/
#ifdef __cplusplus

unsigned long bur_heap_size = 6553500;

#endif

void fSimPIDx(struct fSimPIDx* inst)
{
  BlockIO_SimPIDBR6 *SimPIDBR6_B = &(inst)->bur_BlockIO_SimPIDBR6;
	D_Work_SimPIDBR6 *SimPIDBR6_DWork = &(inst)->bur_D_Work_SimPIDBR6;

  switch (inst->ssMethodType)
  {
   case SS_INITIALIZE:
    /* call model initialize function */
    SimPIDBR6_initialize(SimPIDBR6_DWork, inst);
    break;

   case SS_OUTPUT:
    /* call model step function */
    SimPIDBR6_step(SimPIDBR6_B, SimPIDBR6_DWork, inst);

    break;

   case SS_TERMINATE:
    /* call model terminate function */
    SimPIDBR6_terminate(inst);
    break;
  }
}

/*****************************************************************************
   Function block sample time: 0.01s
 *****************************************************************************/

/*****************************************************************************
   B&R Automation Studio Target for Simulink Version: A4.5.1 (27-Jul-2015)
 *****************************************************************************/

/*======================== TOOL VERSION INFORMATION ==========================*
 * MATLAB 8.0 (R2012b)20-Jul-2012                                             *
 * Simulink 8.0 (R2012b)20-Jul-2012                                           *
 * Simulink Coder 8.3 (R2012b)20-Jul-2012                                     *
 * Embedded Coder 6.3 (R2012b)20-Jul-2012                                     *
 * Stateflow 8.0 (R2012b)20-Jul-2012                                          *
 *============================================================================*/

/*======================= LICENSE IN USE INFORMATION =========================*
 * curve_fitting_toolbox                                                      *
 * matlab                                                                     *
 * matlab_coder                                                               *
 * real-time_workshop                                                         *
 * rtw_embedded_coder                                                         *
 * simulink                                                                   *
 *============================================================================*/
```

#### lib_properties.txt
```
For manual assignment to hardware configuration please
add the following additional include directories:

\Logical\MATLAB_includes\R2012b\

And the following additional build options:

-lm -D MODEL=SimPIDBR6 -D NUMST=1 -D NCSTATES=0 -D HAVESTDIO -D ONESTEPFCN=1 -D TERMFCN=1 -D MAT_FILE=0 -D MULTI_INSTANCE_CODE=1 -D INTEGER_CODE=0 -D MT=0 -D CLASSIC_INTERFACE=0 -D TID01EQ=0
```

### Library Logical/EngineController/Lib_EC/lHiContr (ANSIC)

#### lHiContr.fun
```iecst
FUNCTION_BLOCK HiContr
  VAR_INPUT
    ssMethodType: SINT;
  END_VAR  VAR_INPUT
        MFGainSkipTdown : REAL; (*Gain for MF integrator deloading time in case of skip-fire*)
  END_VAR
  VAR_INPUT
        GIGain : REAL; (*Gain for glow ignition acting on port injection [%*100cycles/events]*)
  END_VAR
  VAR_INPUT
        WCScaling : REAL; (*Scaling relative to Pmax at full load for weak combustion acting on Pmax stability layer offset in optimizer [%/bar]*)
  END_VAR
  VAR_INPUT
        GIPowGain : REAL; (*Gain for glow ignition acting on power reduction [%Pnom*100cycles/events]*)
  END_VAR
  VAR_INPUT
        MFThSkipOn : REAL; (*Threshold for misfire acting on skip fire [events/100cycles]*)
  END_VAR
  VAR_INPUT
        MFThSkipOff : REAL; (*Threshold for skip fire disabling [events/100cycles]*)
  END_VAR
  VAR_INPUT
        PmaxLimReaHys : REAL; (*Hysteresis for detection bit of Pmax limits reached [bar]*)
  END_VAR
  VAR_INPUT
        MFGain : REAL; (*Gain for misfire acting on port injection [%*100cycles /events]*)
  END_VAR
  VAR_INPUT
        WCGain : REAL; (*Gain for weak combustion acting on Pmax stability layer offset in optimizer [bar*100cycles /events]*)
  END_VAR
  VAR_INPUT
        GIThPIDUR : REAL; (*Threshold for glow ignition acting on port injection [events/100cycles]*)
  END_VAR
  VAR_INPUT
        EngStopErrAck : BOOL := FALSE; (*Error acknowledged after engine stopped [boolean]*)
  END_VAR
  VAR_INPUT
        GIContrEnable : BOOL := FALSE; (*Glow ignition control enabled [boolean]*)
  END_VAR
  VAR_INPUT
        GIPIDURLimMin : REAL; (*Minimum limit for glow ignition acting on port injection [%ofPIDURglobal]*)
  END_VAR
  VAR_OUTPUT
        PIDUROffsetGI : REAL; (*PIDUR offset from glow ignition [% PIDUR global]*)
  END_VAR
  VAR_INPUT
        MFPIDURLimMax : REAL; (*Maximum limit for misfire acting on port injection [%PIDURglobal]*)
  END_VAR
  VAR_INPUT
        MFThPIDUR : REAL; (*Threshold for misfire acting on port injection duration [events/100cycles]*)
  END_VAR
  VAR_INPUT
        MFContrEnable : BOOL := FALSE; (*Misfire control enabled [boolean]*)
  END_VAR
  VAR_OUTPUT
        PIDUROffsetMF : REAL; (*PIDUR offset from misfire [% PIDUR global]*)
  END_VAR
  VAR_OUTPUT
        MFIntOut : REAL; (*Misfire integrator output [events/100 cycles]*)
  END_VAR
  VAR_OUTPUT
        WCIntOut : REAL; (*Weak combustion integrator output [events/100 cycles]*)
  END_VAR
  VAR_OUTPUT
        GIIntOut : REAL; (*Glow ignition integrator output [events/100 cycles]*)
  END_VAR
  VAR_INPUT
        PmaxLimContrEnable : BOOL := FALSE; (*Pmax limit control enabled [boolean]*)
  END_VAR
  VAR_INPUT
        PmaxLimDiane : REAL; (*Pmax limit parameter from Diane [bar]*)
  END_VAR
  VAR_INPUT
        PmaxSDLimMar : REAL; (*Margin to Pmax Shutdown Limit [bar]*)
  END_VAR
  VAR_INPUT
        PmaxStdevFact : REAL; (*Pmax standard deviation factor []*)
  END_VAR
  VAR_INPUT
        PmaxContrGain : REAL; (*Pmax controller gain [%PIDUR/bar]*)
  END_VAR
  VAR_INPUT
        PmaxContrLimMin : REAL; (*Minimum PIDUR offset set by Pmax limiting controller [%PIDUR]*)
  END_VAR
  VAR_OUTPUT
        PIDUROffsetPmax : REAL; (*Pmax limit controller output [% PIDUR global]*)
  END_VAR
  VAR_INPUT
        GIThSkipReset : REAL; (*Reset threshold for glow ignition acting on skip-fire [events/100cycles]*)
  END_VAR
  VAR_OUTPUT
        GICountOut : REAL; (*Glow ignition counter output [counts]*)
  END_VAR
  VAR_OUTPUT
        PmaxAv : REAL; (*Pmax moving average [bar]*)
  END_VAR
  VAR_OUTPUT
        PmaxStd : REAL; (*Pmax moving standard deviation [bar]*)
  END_VAR
  VAR_INPUT
        WCThPmax : REAL; (*Threshold for weak combustion acting on Pmax stability layer offset in optimizer [events/100cycles]*)
  END_VAR
  VAR_INPUT
        GIThSkip : REAL; (*Threshold for glow ignition acting on skip-fire [events/100cycles]*)
  END_VAR
  VAR_INPUT
        GIThCount : REAL; (*Threshold for number of task cycles showing glow ignition to activate power reduction [number of task cycles]*)
  END_VAR
  VAR_INPUT
        Misfire2 : BOOL := FALSE; (*Late misfire [boolean]*)
  END_VAR
  VAR_INPUT
        Misfire1 : BOOL := FALSE; (*Early misfire [boolean]*)
  END_VAR
  VAR_INPUT
        SensSignFault : BOOL := FALSE; (*Sensor signal fault [boolean]*)
  END_VAR
  VAR_INPUT
        TGICount : REAL; (*Glow ignition upwards integration time [combustion cycles]*)
  END_VAR
  VAR_INPUT
        TdownGI : REAL; (*Glow ignition downwards integration time [combustion cycles]*)
  END_VAR
  VAR_INPUT
        GlowIgn : BOOL := FALSE; (*Glow ignition [boolean]*)
  END_VAR
  VAR_INPUT
        TupGI : REAL; (*Glow ignition upwards integration time [combustion cycles]*)
  END_VAR
  VAR_INPUT
        TdownMF : REAL; (*Misfire downwards integration time [combustion cycles]*)
  END_VAR
  VAR_INPUT
        WCPmaxLimMax : REAL; (*Maximum limit for weak combustion acting on Pmax stability layer offset in optimizer [%ofPmax]*)
  END_VAR
  VAR_INPUT
        TupWC : REAL; (*Weak combustion upwards integration time [combustion cycles]*)
  END_VAR
  VAR_INPUT
        TupMF : REAL; (*Misfire upwards integration time [combustion cycles]*)
  END_VAR
  VAR_INPUT
        TdownWC : REAL; (*Weak combustion downwards integration time [combustion cycles]*)
  END_VAR
  VAR_INPUT
        KnockCountMeasAct : BOOL := FALSE; (*Knock countermeasures currently active [boolean]*)
  END_VAR
  VAR_INPUT
        SkipCylExt : BOOL := FALSE; (*External skip-fire command*)
  END_VAR
  VAR_INPUT
        WCContrEnable : BOOL := FALSE; (*Weak combustion control enabled [boolean]*)
  END_VAR
  VAR_OUTPUT
        FaultMFSign : BOOL := FALSE; (*Faulty misfire detection*)
  END_VAR
  VAR_OUTPUT
        MFB50Freeze : BOOL := FALSE; (*Command to freeze MFB50% controller*)
  END_VAR
  VAR_OUTPUT
        OptPIDFreeze : BOOL := FALSE; (*Command to freeze optimizer PIDs*)
  END_VAR
  VAR_OUTPUT
        PIDUROffsetCyl : REAL; (*PI duration offset for cylinder*)
  END_VAR
  VAR_OUTPUT
        PmaxStabLayOffset : REAL; (*Pmax stability layer offset [% Pmax]*)
  END_VAR
  VAR_OUTPUT
        PmaxLimReached : BOOL := FALSE; (*Pmax limit reached*)
  END_VAR
  VAR_OUTPUT
        SkipCyl : BOOL := FALSE; (*Cylinder to be skipped*)
  END_VAR
  VAR_OUTPUT
        PowRedCyl : REAL; (*Power reduction for cylinder*)
  END_VAR
  VAR_INPUT
        Pmax : REAL; (*Peak firing pressure average [bar]*)
  END_VAR
	VAR
		bur_HiContr_DWork : D_Work_HiContr;
	END_VAR
	VAR
		bur_HiContr_B : BlockIO_HiContr;
	END_VAR
END_FUNCTION_BLOCK
```

#### lHiContr.typ
```iecst
 TYPE

END_TYPE
TYPE
	D_Work_HiContr : STRUCT

		DiscreteTimeIntegrator_DSTATE : REAL;
		DiscreteTimeIntegrator_DSTATE_e : REAL;
		DiscreteTimeIntegrator_DSTATE_c : REAL;
		TappedDelaysetasN_cyc_X : ARRAY[0..99] OF REAL;
		DiscreteTimeIntegrator_DSTATE_n : REAL;
		DiscreteTimeIntegrator_PrevRese : SINT;
		DiscreteTimeIntegrator_PrevRe_f : SINT;
		DiscreteTimeIntegrator_PrevRe_c : SINT;
		DiscreteTimeIntegrator_PrevRe_n : SINT;
		Relay1_Mode : BOOL;
		Relay_Mode : BOOL;
	END_STRUCT;

	 BlockIO_HiContr : STRUCT

		Input17 : REAL;
		DiscreteTimeIntegrator : REAL;
		Input13 : REAL;
		Switch2 : REAL;
		Input11 : REAL;
		Input14 : REAL;
		DiscreteTimeIntegrator_d : REAL;
		Switch2_e : REAL;
		DiscreteTimeIntegrator_l : REAL;
		Input11_h : REAL;
		Input7 : REAL;
		Divide : REAL;
		Sqrt : REAL;
		Input8 : REAL;
		Input9 : REAL;
		Input10 : REAL;
		Switch2_k : REAL;
		Input19 : REAL;
		DiscreteTimeIntegrator_dl : REAL;
		Input16 : REAL;
		Input18 : REAL;
		Input21 : REAL;
		Input6 : REAL;
		GIPowGainPnom100cyclesevents : REAL;
		Input5 : REAL;
		Input4 : REAL;
		Input1 : REAL;
		Input12 : REAL;
		Input2 : REAL;
		Input20 : REAL;
		Input3 : REAL;
		Switch2_a : REAL;
		Switch4 : REAL;
		Input3_g : REAL;
		Input5_c : BOOL;
		Input9_a : BOOL;
		Input7_c : BOOL;
		Input10_h : BOOL;
		Input1_h : BOOL;
		Input20_o : BOOL;
		Input4_d : BOOL;
		Input2_g : BOOL;
		Input6_a : BOOL;
		Compare : BOOL;
		LogicalOperator13 : BOOL;
		Input12_e : BOOL;
		LogicalOperator2 : BOOL;
		Input8_f : BOOL;
		LogicalOperator7 : BOOL;
		LogicalOperator8 : BOOL;
	END_STRUCT;

END_TYPE
```
